//报警复位
IF machine.reset THEN
  MEMSET(ADR(machine.presetAlarms),0,SIZEOF(machine.presetAlarms));
  MEMSET(ADR(machine.userAlarms),0,SIZEOF(machine.userAlarms));
  machine.publicAlarm := FALSE;
  machine.report.alarming := FALSE;
  machine.report.stationAlarming := FALSE;
END_IF;

// 报警顶栏显示
IF NOT alarmingCache AND  machine.alarming THEN
  machine.alarmTopBarDisplay := TRUE;
ELSIF NOT machine.alarming THEN
  machine.alarmTopBarDisplay := FALSE;
END_IF;
alarmingCache :=  machine.alarming;

//复位按钮灯
machine.alarmCanReset := machine.report.alarmCanReset;

machine.resetButtonLight := machine.lampTesthmi        //指示灯测试
OR (NOT machine.alarmCanReset AND machine.alarming) //报警中常亮
OR (machine.alarmCanReset AND clock.c1s);           //报警可复位闪烁
machine.alarmCanReset := FALSE;
machine.report.alarmCanReset := FALSE;
END_ACTION

ACTION AutoTip:
//--------------------------AutoTip---------------------------//
  
//机器未初始化
machine.presetAutoTips[0] := NOT machine.initDone;
//机器运行条件不足
machine.presetAutoTips[1] := NOT machine.runPermit;

//整机自动提示
machine.autoTip :=
FUN_AryBitCount_RD(machine.presetAutoTips) >0
OR FUN_AryBitCount_RD(machine.userAutoTips) >0
OR machine.report.autoTip
OR machine.report.stationAutoTip;
machine.report.autoTip := FALSE;
machine.report.stationAutoTip := FALSE; 

//自动提示弹窗
IF machine.autoTip AND machine.start THEN
  machine.autoTipTrigger := TRUE;
  machine.popup := POPUP_AUTO_TIP;
END_IF;
IF machine.popup = 0 THEN
  machine.autoTipTrigger := FALSE;
END_IF;
END_ACTION

ACTION CycleTime:
//--------------------------CycleTime---------------------------//
//机器周期计时,
IF machine.cycleTimeEnd THEN
  machine.cycleTime :=TIME_TO_DINT( cycleTimeTimer.ET);
END_IF;
cycleTimeTimer(IN := machine.cycleTimeStart AND NOT (machine.cycleTimeEnd OR machine.initing),
               PT := T#10M
);
machine.cycleTimeEnd := FALSE;
END_ACTION

ACTION Empty:
//--------------------------Empty---------------------------//
  
//清料条件
emptyPermit := machine.eStop
AND machine.initDone
AND NOT machine.initing;

// 清料完成，延时复位完成信号
IF machine.emptyDone
  AND NOT machine.emptying   //确保清料中断开
  AND NOT machine.running    //确保自动中断开
THEN
  machine.emptyDone := FALSE;
END_IF;

// 清料hmi，弹出清料确认对话框
IF emptyPermit
  AND machine.emptyhmi
THEN
  machine.popup := POPUP_EMPTY_CONFIRM;
END_IF;
// 清料中
IF NOT machine.initing
  AND NOT machine.emptyDone
THEN
  IF machine.emptyConfirm
    AND emptyPermit
  THEN
    machine.emptying := TRUE;
  END_IF;
  
ELSE
  machine.emptying := FALSE;
END_IF;

// 不在清料中且清料完成，弹出清料完成对话框
// 清料完成信号由功能块外部判断清料完成后置位，功能块内部不进行置位
IF NOT machine.emptying
  AND machine.emptyDone
THEN
  machine.popup := POPUP_EMPTY_DONE;
END_IF;
END_ACTION

ACTION Flow:
//--------------------------Flow---------------------------//
//流程监控
FOR index := 0 TO flowNum DO
  IF machine.flow[index].actStep = 999 THEN
    machine.flow[index].uninterrupted := TRUE;
  END_IF;
  //流程上一步记录
  IF machine.flow[index].actStep <> flowStepCache[index] THEN
    machine.flow[index].prevStep := flowStepCache[index];
  END_IF;
  flowStepCache[index] := machine.flow[index].actStep;
  //流程超时计时
flowTimeoutTimer[index](IN := machine.flow[index].timeoutEnable
            AND NOT machine.flow[index].timeoutException
            AND (machine.running OR machine.initing)
            AND machine.flow[index].actStep > 0
            AND machine.flow[index].actStep = flowStepCache[index],
            PT := machine.flow[index].setTimeout,
		  Q=>);
  machine.flow[index].timeoutException := FALSE;
  //流程超时报警置位
IF flowTimeoutTimer[index].Q THEN
    machine.flow[index].timeoutAlarm := TRUE;
    machine.presetAlarms[index + 8] := TRUE;
  ELSIF machine.reset THEN
    machine.flow[index].timeoutAlarm := FALSE;
  END_IF;
END_FOR;
END_ACTION

ACTION General:
//--------------------------General---------------------------//
FUN_UpdateLeftSidebar_RD(machine:=machine,
			  				hmi:=hmi);

//  触摸屏按钮
machine.start := machine.startButton OR hmi.button.start OR machine.starthmi;
machine.stop := machine.stopButton OR hmi.button.stop OR machine.stophmi;
machine.reset := machine.resetButton OR hmi.button.reset OR machine.resethmi;
machine.pause := machine.pauseButton OR hmi.button.pause OR machine.pausehmi;
machine.init := machine.initButton OR hmi.button.init OR machine.inithmi;
manualSwitch := machine.manualSwitch OR hmi.button.manualSwitch;
autoSwitch := machine.autoSwitch OR hmi.button.autoSwitch;
IF manualSwitch OR autoSwitch THEN
  manualModehmi := FALSE;   //实体手自动旋钮复位hmi
  autoModehmi := FALSE;
END_IF;

IF NOT manualModehmiCache AND machine.manualModehmi THEN
	autoModehmi := FALSE;
	manualModehmi := NOT manualModehmi;
END_IF;
manualModehmiCache := machine.manualModehmi;

IF  NOT autoModehmiCache AND machine.autoModehmi THEN
	autoModehmi := NOT autoModehmi;
	manualModehmi := FALSE;
END_IF;
autoModehmiCache := machine.autoModehmi;

//手动模式
machine.manualMode := NOT machine.jogMode
AND (manualSwitch AND NOT autoSwitch
OR NOT manualSwitch AND NOT autoSwitch
AND manualModehmi AND NOT autoModehmi
);
//自动模式
machine.autoMode := NOT machine.jogMode
AND (NOT manualSwitch AND autoSwitch
OR NOT manualSwitch AND NOT autoSwitch
AND NOT manualModehmi AND autoModehmi
);

IF machine.manualMode THEN
  machine.mode := MANUAL_MODE;
ELSIF machine.autoMode THEN
  machine.mode := AUTO_MODE;
ELSE
  machine.mode := UNDEFINED_MODE;
END_IF;

// 三色灯
machine.greenStatusLight := machine.lampTesthmi OR (machine.running AND NOT machine.alarming);
machine.yellowStatusLight := machine.lampTesthmi OR (NOT machine.running AND NOT machine.alarming);
machine.redStatusLight := machine.lampTesthmi OR machine.alarming;
machine.buzzer := machine.alarming AND NOT buzzerTimer.Q;
buzzerTimer(IN := machine.alarming,
             PT := machine.buzzerTime);
END_ACTION

ACTION Init:
//--------------------------Init---------------------------//
// 初始化条件
initPermit := safePermit
AND machine.manualMode
AND NOT machine.alarming;

//初始化确认弹窗
IF machine.init THEN
  IF machine.alarming THEN
    machine.popup := POPUP_INIT_ALARM;
  ELSIF initPermit AND NOT machine.initing THEN
    machine.popup := POPUP_INIT_FAILED;
  END_IF;
END_IF;

 //整机初始化完成
machine.initDone := initDoneTimer.Q
												AND NOT machine.initConfirm
												AND machine.initFlowDone
												AND NOT machine.report.stationNotInitDone;

// 初始化中
IF initPermit
  AND NOT machine.pause
  AND NOT machine.initDone
AND FUN_AryBitCount_RD(machine.userManualTips) =0
THEN
  IF initConfirmCache AND NOT machine.initConfirm THEN
    machine.initing := TRUE;
  END_IF;
ELSE
  machine.initing := FALSE;
END_IF;
initConfirmCache := machine.initConfirm ;  // 初始化确认下降沿

// 初始化延时
initTimer(IN := machine.initing,
           PT := T#10S,
           Q  => );

// 初始化完成延时
initDoneTimer(IN := NOT machine.initConfirm,
               PT := T#10S,
			 Q=>);

// 初始化超时
initTimeoutTimer(IN := machine.initing,
                  PT := machine.initTimeout);

// 初始化按钮灯，初始化中常亮  
machine.initButtonLight := machine.lampTesthmi OR machine.initing;
  
machine.report.stationNotInitDone := FALSE;

 //整机初始化中下降沿
IF  initingCache AND NOT machine.initing THEN
  IF  machine.alarming THEN			// 初始化中报警对话框
    machine.popup := POPUP_INITING_ALARM;	
	ELSIF machine.initDone THEN		// 初始化完成对话框
    machine.popup := POPUP_INIT_DONE;	  
	ELSE												// 初始化失败对话框
    machine.popup := POPUP_INIT_CONFIRM;
  END_IF;	  
END_IF;
initingCache:=machine.initing;
END_ACTION

ACTION LeftSidebar:
//--------------------------LeftSidebar---------------------------//
  //左侧边栏按钮控制

//---------------------------

hmi.button.startLight := machine.startButtonLight;
hmi.button.stopLight := machine.stopButtonLight;
hmi.button.resetLight :=machine.resetButtonLight;
hmi.button.pauseLight :=   machine.pauseButtonLight;
hmi.button.initLight := machine.initButtonLight;
END_ACTION

ACTION ManualTip:
//--------------------------ManualTip---------------------------//
  
// 复位手动提示
IF machine.reset OR Hmi.machineHmi.tipReset THEN
  machine.tipReset := TRUE;
END_IF;
IF machine.tipReset THEN
  MEMSET(ADR(machine.presetAutoTips),0,SIZEOF(machine.presetAutoTips));
  MEMSET(ADR(machine.userAutoTips),0,SIZEOF(machine.userAutoTips));
  MEMSET(ADR(machine.presetManualTips),0,SIZEOF(machine.presetManualTips));
  MEMSET(ADR(machine.userManualTips),0,SIZEOF(machine.userManualTips));	
  //复位提示窗口
  IF machine.popup = 0 THEN
 Hmi.machineHmi.tipReset:=FALSE;	
    machine.tipReset := FALSE; 
  ELSE
    machine.popup := 0;
  END_IF;
END_IF;

//机器手动提示
IF machine.start OR machine.init THEN
  machine.presetManualTips[0] := NOT machine.eStop;     //急停中,无法操作
  machine.presetManualTips[1] := NOT machine.safety;    //安全条件不满足,无法操作
  machine.presetManualTips[2] := NOT machine.allDoorClosed;  //安全门未锁好,无法操作
  machine.presetManualTips[3] := NOT machine.airOn;     //气压不足,无法操作
  IF machine.init THEN
    machine.presetManualTips[4] := NOT machine.manualMode;//不在手动模式,无法操作
  ELSIF machine.start THEN
    machine.presetManualTips[5] := NOT machine.autoMode;  //不在自动模式,无法操作
  END_IF;
END_IF;

//机器手动提示中
machine.manualTip :=
FUN_AryBitCount_RD(machine.presetManualTips) >0
OR FUN_AryBitCount_RD(machine.userManualTips) >0
OR machine.report.stationManualTip
OR machine.report.manualTip;
machine.report.manualTip := FALSE;
machine.report.stationManualTip := FALSE;

// 手动提示弹窗
IF machine.manualTip THEN
  machine.popup := POPUP_MANUAL_TIP;
END_IF;
END_ACTION

ACTION Paused:
//--------------------------Paused---------------------------//
// 暂停中
IF machine.pause THEN
  machine.paused := TRUE;
END_IF;

// 急停、初始化、启动，复位暂停中
IF NOT machine.eStop
  OR machine.initing
  OR machine.start
THEN
  machine.paused := false;
END_IF;

// 暂停按钮灯，暂停中常亮
machine.pauseButtonLight := machine.lampTesthmi  OR machine.paused;
END_ACTION

ACTION Safety:
//--------------------------Safety---------------------------//
  
//急停就绪    
machine.eStop := NOT machine.report.notEstops;
machine.report.notEstops := FALSE;

//安全门就绪 
// machine.allDoorClosed := NOT machine.report.notSafetyDoors;
machine.report.notSafetyDoors := FALSE;

safePermit := machine.eStop
AND machine.allDoorClosed
AND machine.airOn
AND machine.safety;
END_ACTION

ACTION SetUp:
//--------------------------SetUp---------------------------//

  
IF NOT activated THEN
	  activated:=TRUE;
	//赋初始值
	machine.runPermit			:=TRUE;
	machine.startPermit			:=TRUE;
	machine.mainScreenNo 		:= 10; //自定义主画面显示
	machine.initTimeout			:= T#60s; // 初始化超时时间
	machine.idealCycleTime 		:= t#2s;  //理想周期时间
	machine.stopTimeout			:= T#4s; //停止超时时间,理想周期2倍以上时间
	machine.buzzerTime			:= T#3s; // 蜂鸣器持续时间
	machine.requestCountdown 	:=UINT#10;  // HMI请求控制权倒计时
	machine.sidebar.typeData[1]:=1;
	machine.sidebar.typeData[2]:=2;
	machine.sidebar.typeData[5]:=3;
    //流程数量
	flowNum := SIZEOF(machine.flow) -1;
	FOR index:=0 TO flowNum DO
		//machine.flow[index].timeoutEnable	:=FALSE;
	    machine.flow[index].setTimeout			:=T#30s;
	END_FOR;
	
END_IF;
machine.sidebar.typeData[1]:=1;
machine.sidebar.typeData[2]:=2;
machine.sidebar.typeData[5]:=3;
END_ACTION

ACTION Start:
//--------------------------Start---------------------------//
// 运行条件
machine.ready := safePermit
AND machine.runPermit
AND machine.initDone
AND (machine.autoMode OR machine.jogMode)
AND NOT machine.alarming
AND NOT machine.autoTip;
// 运行中
IF machine.ready
  AND NOT machine.pause
  AND NOT machine.paused
  AND NOT machine.stopDone
  AND NOT machine.emptyDone
THEN
  IF machine.autoMode THEN
    IF machine.start
      AND NOT machine.reset
      AND NOT machine.stop
    THEN     //自动模式下按下启动按钮自动中保持
      machine.running := TRUE;
    END_IF;
  ELSIF machine.jogMode
    AND NOT machine.reset
    AND NOT machine.stop
    AND machine.start
  THEN
    machine.running := TRUE;  //寸动模式下按下启动按钮自动中，抬起按钮复位自动中
  ELSE
    machine.running := FALSE;
  END_IF;
ELSE
  machine.running := FALSE;
END_IF;

// 启动按钮灯，运行中常亮，准备就绪时闪烁

machine.startButtonLight := machine.lampTesthmi
OR machine.running
OR (machine.ready AND clock.c1s);
END_ACTION

ACTION Stop:
//--------------------------Stop---------------------------//
// 自动中按停止，置位停止中
IF (machine.stop OR machine.alarming)
  AND NOT machine.stopDone
  AND NOT machine.paused
THEN
  machine.stopping := TRUE;
END_IF;

// 急停，初始化，启动，暂停，停止完成且不在自动中，复位停止中
IF NOT machine.eStop
  OR machine.initing
  OR machine.start
  OR machine.pause
  OR machine.stopDone
  AND NOT machine.running
THEN
  machine.stopping := FALSE;
END_IF;

//停止完成
stopTimer(IN := machine.stopping,
           PT := machine.stopTimeout);
IF machine.stopping AND (machine.stopDoneAllow OR stopTimer.Q) THEN
  machine.stopDone := TRUE;
ELSIF NOT machine.eStop
  OR machine.initing
  OR machine.start
  OR machine.pause
THEN
  machine.stopDone := FALSE;
END_IF;

// 停止按钮灯，停止完成常亮，停止中闪烁
  machine.stopButtonLight := machine.lampTesthmi
OR machine.stopDone
OR (machine.stopping AND clock.c1s);
END_ACTION

ACTION Tip:
//--------------------------Tip ---------------------------//
  
IF machine.alarming THEN
  machine.status := ALARMING;
ELSIF machine.initing THEN
  machine.status := INITING;
ELSIF machine.running THEN
  machine.status := RUNNING;
ELSIF machine.ready THEN
  machine.status := READY;
ELSE
  machine.status := 0;
END_IF;

machine.presetTips[1] := machine.alarming;
machine.presetTips[2] := machine.paused;
machine.presetTips[3] := machine.stopping;
machine.presetTips[4] := machine.initing;
machine.presetTips[5] := machine.running;
machine.presetTips[6] := machine.ready AND NOT machine.running;
machine.presetTips[7] := NOT machine.ready;
machine.presetTips[10] := machine.emptying;
machine.presetTips[11] := machine.emptyDone;
machine.presetTips[21] := machine.dryRun;
END_ACTION

END_FUNCTION_BLOCK

// ---- Standard/FUN/FUN_UpdateLeftSidebar_RD.TcPOU
FUNCTION FUN_UpdateLeftSidebar_RD : bool
VAR_IN_OUT
machine       : UDT_Machine_RD;
hmi           : UDT_hmi_RD;
END_VAR
VAR CONSTANT
LEFT_SIDEBAR_MANUAL_MODE : INT :=1;
LEFT_SIDEBAR_AUTO_MODE   : INT :=2;
LEFT_SIDEBAR_JOG_MODE    : INT :=3;
LEFT_SIDEBAR_SETUP_MODE  : INT :=4;
LEFT_SIDEBAR_INIT        : INT :=5;
LEFT_SIDEBAR_START       : INT :=6;
LEFT_SIDEBAR_STOP        : INT :=7;
LEFT_SIDEBAR_RESET       : INT :=8;
LEFT_SIDEBAR_EMPTY       : INT :=9;
LEFT_SIDEBAR_PAUSE       : INT :=10;
LEFT_SIDEBAR_MANUAL      : INT :=11;
LEFT_SIDEBAR_PARAMETER   : INT :=12;
LEFT_SIDEBAR_STATION     : INT :=13;

END_VAR

// 获取左侧边栏按钮是否按下
machine.manualModeHmi := machine.sidebar.click[LEFT_SIDEBAR_MANUAL_MODE];
machine.autoModeHmi := machine.sidebar.click[LEFT_SIDEBAR_AUTO_MODE];
machine.jogModeHmi := machine.sidebar.click[LEFT_SIDEBAR_JOG_MODE];
machine.setupModeHmi := machine.sidebar.click[LEFT_SIDEBAR_SETUP_MODE];
machine.initHmi := machine.sidebar.click[LEFT_SIDEBAR_INIT];
machine.startHmi := machine.sidebar.click[LEFT_SIDEBAR_START];
machine.stopHmi := machine.sidebar.click[LEFT_SIDEBAR_STOP];
machine.resetHmi := machine.sidebar.click[LEFT_SIDEBAR_RESET];
machine.emptyHmi := machine.sidebar.click[LEFT_SIDEBAR_EMPTY];
machine.pauseHmi := machine.sidebar.click[LEFT_SIDEBAR_PAUSE];
IF machine.sidebar.click[LEFT_SIDEBAR_MANUAL] THEN
	hmi.toManualPageClick:=TRUE;
END_IF;
IF machine.sidebar.click[LEFT_SIDEBAR_PARAMETER] THEN
	hmi.toParameterPageClick:=TRUE;
END_IF;
IF machine.sidebar.click[LEFT_SIDEBAR_STATION] THEN
	hmi.toStationPageClick:=TRUE;
END_IF;

// 设置左侧边栏按钮状态显示
machine.sidebar.status[LEFT_SIDEBAR_MANUAL_MODE] := machine.manualMode;
machine.sidebar.status[LEFT_SIDEBAR_AUTO_MODE] := machine.autoMode;
machine.sidebar.status[LEFT_SIDEBAR_JOG_MODE] := machine.jogMode;
machine.sidebar.status[LEFT_SIDEBAR_SETUP_MODE] := machine.setupMode;
machine.sidebar.status[LEFT_SIDEBAR_INIT] := machine.initButtonLight;
machine.sidebar.status[LEFT_SIDEBAR_START] := machine.startButtonLight;
machine.sidebar.status[LEFT_SIDEBAR_STOP] := machine.stopButtonLight;
machine.sidebar.status[LEFT_SIDEBAR_RESET] := machine.resetButtonLight;
machine.sidebar.status[LEFT_SIDEBAR_EMPTY] := machine.emptying;
machine.sidebar.status[LEFT_SIDEBAR_PAUSE] := machine.pauseButtonLight;
machine.sidebar.status[LEFT_SIDEBAR_MANUAL] := hmi.inManualPage;
machine.sidebar.status[LEFT_SIDEBAR_PARAMETER] := hmi.inParameterPage;
machine.sidebar.status[LEFT_SIDEBAR_STATION] := hmi.inStationPage;

END_FUNCTION

// ---- Standard/Unit/03 Estop/FB_Estop_RD.TcPOU
FUNCTION_BLOCK FB_Estop_RD
VAR_IN_OUT
vari         : UDT_Estop_RD;
machine      : UDT_Machine_RD;

END_VAR
VAR
resetCache      : BOOL;
END_VAR

//急停复位
IF machine.reset AND NOT resetCache AND vari.input THEN
	vari.notEstop:=FALSE;
END_IF;

//急停
IF NOT vari.disable AND NOT vari.input THEN
	Vari.notEstop:=TRUE;
	machine.report.notEstops:=TRUE;
END_IF;

resetCache:=machine.reset;

END_FUNCTION_BLOCK

// ---- Standard/Unit/04 SafetyDoor/FB_SafetyDoor_RD.TcPOU
FUNCTION_BLOCK FB_SafetyDoor_RD
VAR_IN_OUT
machine : UDT_Machine_RD; //
vari : UDT_SafetyDoor_RD; //
clock : UDT_Clock_RD; //
END_VAR

VAR
prohibit : BOOL; // 禁止解锁
unlockButtonCache : Bool; // 解锁按钮缓存
permitTimer : TON; // 解锁许可延时
autoLockTimer : TON; // 自锁延时

END_VAR

VAR CONSTANT
NOT_LOCKED      : UINT:=1;
DISABLED        : UINT:=2;
END_VAR

  //================================================================================== 
  // Harmontromics / (C) Copyright (2021) 
  //----------------------------------------------------------------------------------
  // Title:               Safety Door
  // Comment/Function:    实现安全门的控制，自/手动上锁、按钮解锁
  // Library/Family:      (that the source is dedicated to)
  // Author:              David.Wong
  // Target System: 
  // Engineering:         Sysmac Studio
  // Restrictions:        (OB types, etc.)
  // Requirements:        (hardware, technological package, etc.) 
  //----------------------------------------------------------------------------------
  // Change log table:
  // Version     | Date       | Expert in charge | Changes applied
  //-------------|------------|------------------|------------------------------------
  // 001.000.000 | 2021-12-11 | David.Wong       | First released version
  //             |            |                  | 
  //             |            |                  |              
  //             |            |                  | 
  //================================================================================== 
SetUp();
SafetyDoor();
Tip();

ACTION SafetyDoor:
//------------------------------SafetyDoor-------------------------------------//
  
//  禁止解锁
prohibit := machine.eStop
AND vari.inputLocked
AND (NOT machine.manualMode
OR machine.initing
OR machine.running
OR vari.prohibitUnlock);

//  解锁许可延时
permitTimer(
	IN:=NOT Prohibit,
	PT:=T#500MS,
	Q=> , ET=> 
);
  
//  插销没到位且没锁好信号时自动弹开
IF vari.inputUnlockButton
	AND
	permitTimer.Q	  
	//AND NOT vari.inputLocked   
	//AND NOT vari.inputArrived
THEN
  vari.outputLockCoil := TRUE;
END_IF;

//  解锁按钮操作，自动上锁时解锁，非自动上锁时解锁和上锁
IF NOT unlockButtonCache AND vari.inputUnlockButton THEN
  vari.outputLockCoil := NOT vari.outputLockCoil AND NOT vari.autoLock;
END_IF;
unlockButtonCache := vari.inputUnlockButton;

//  自锁延时
autoLockTimer(IN := vari.autoLock AND NOT vari.inputUnlockButton,
			  PT := vari.autoLockTime
);  
  
//  自动上锁及禁止解锁
IF vari.inputArrived
  AND
  (autoLockTimer.Q
  OR NOT permitTimer.Q)
THEN
  vari.outputLockCoil := FALSE;
END_IF;

//  解锁按钮灯输出
IF vari.inputLocked THEN
  vari.outputUnlockButtonLight := vari.lightWhenLocked;
ELSE
  vari.outputUnlockButtonLight := clock.c1s;
END_IF;
END_ACTION

ACTION SetUp:
//------------------------------SetUp-------------------------------------//
  IF machine.startUp THEN
    IF vari.name[machine.actLanguage] <> '' THEN
      vari.name[0] := vari.name[machine.actLanguage];
    END_IF;
	vari.autoLockTime:=T#3s;
  END_IF;
END_ACTION

ACTION Tip:
//------------------------------Tip---------------------------------------------//
  
// 安全门未锁好提示
IF (NOT vari.inputArrived
  OR NOT vari.inputLocked
  OR NOT vari.outputLockCoil)
  AND NOT vari.disabled
THEN
  vari.notLocked := TRUE; // 安全门未锁好报警
ELSIF machine.reset THEN
  vari.notLocked := FALSE;
END_IF;

//反馈安全没锁好
IF vari.notLocked THEN
  machine.report.notSafetyDoors := TRUE;
END_IF;
END_ACTION

END_FUNCTION_BLOCK

// ---- Standard/Unit/07 Sensor/FB_Sensor_RD.TcPOU
FUNCTION_BLOCK FB_Sensor_RD
VAR_IN_OUT
machine : UDT_Machine_RD; //
station : UDT_Station_RD; //
vari : UDT_SensorVar_RD; //
data : UDT_SensorData_RD; //
END_VAR
VAR_OUTPUT
END_VAR
VAR
inputCache : BOOL; //
checkCache : Bool; //
resetCache : Bool; //
onTimer : TON; //
offTimer : TON; //
flickerTimer : TON; //
firstCall    : BOOL :=TRUE;

END_VAR

SetUp();
Delay();
Alarm();

ACTION Alarm:
//-------------------------------Alarm--------------------------//
  
//复位报警并计数清零
IF NOT resetCache AND machine.reset THEN
  IF vari.unchangeError THEN
    vari.count := 0;
    vari.unchangeError := FALSE;
  END_IF;
  vari.flickerError := FALSE;
END_IF;
resetCache := machine.reset;
  
vari.alarming := vari.unchangeError
OR vari.flickerError;

//反馈上一级报警中
IF vari.alarming THEN
  station.report.alarming := TRUE;
  machine.alarmCount := machine.alarmCount +1;
END_IF;
END_ACTION

ACTION Delay:
//-----------------------------------Delay--------------------------//
//屏蔽传感器时,ON OFF都输出
IF NOT data.disabled THEN
  onTimer(IN := vari.input,
           PT :=UDINT_TO_TIME(data.onTime),
           Q => vari.isOn);
  offTimer(IN := NOT vari.input,
            PT := UDINT_TO_TIME(data.offTime),
            Q => vari.isOff);
  IF inputCache <> vari.input OR data.setCount = 0 THEN//输入有变化或设置值0清空计数
    vari.count := 0;
  ELSIF NOT checkCache AND vari.check THEN    //check上升沿计数+1
    vari.count :=vari.count + 1;
  ELSIF checkCache AND NOT vari.check       //check下降沿且计数计数值大于等于设定值时报警
    AND vari.count >= data.setCount
  THEN
    vari.unchangeError := TRUE;
  END_IF;
  
  //超过On、Off延时之和2倍时间都没到位报警传感器闪烁异常
  data.flickerTime := MAX(data.flickerTime,(data.onTime + data.offTime) * 2);
  flickerTimer(IN := NOT vari.isOn AND NOT vari.isOff,
               PT := UDINT_TO_TIME(data.flickerTime)
			   );
  
  inputCache := vari.input;
  checkCache := vari.check;
ELSE
  vari.isOn := TRUE;
  vari.isOff := TRUE;
  vari.count := 0;
END_IF;
END_ACTION

ACTION SetUp:
//开机或切换语言后执行一个扫描周期
//------------------------------------ SetUp--------------------------//
  IF firstCall THEN
    // 显示在HMI上面
    vari.display := TRUE;
	firstCall :=FALSE;
  END_IF;
END_ACTION

END_FUNCTION_BLOCK

// ---- Standard/Unit/12 Delay/FB_Delay_RD.TcPOU
FUNCTION_BLOCK FB_Delay_RD
VAR_IN_OUT
machine : UDT_Machine_RD; //
station : UDT_Station_RD; //
vari : UDT_DelayVar_RD; //
data : UDT_DelayData_RD; //
END_VAR
VAR_OUTPUT
END_VAR

VAR
timer1    : TON;
END_VAR

timer1(IN := vari.input AND vari.actTime <= data.setTime,
	         PT := data.setTime,
	         ET => vari.actTime,
	         Q => vari.isOn);
IF vari.isOn OR vari.actTime > data.setTime THEN
  vari.input := FALSE;
END_IF;

END_FUNCTION_BLOCK

// ---- Standard/Unit/08 Motor/FB_Motor_RD.TcPOU
FUNCTION_BLOCK FB_Motor_RD
VAR_IN_OUT
machine   : UDT_Machine_RD;
station   : UDT_Station_RD;
vari      : UDT_MotorVar_RD;
data      : UDT_MotorData_RD;
END_VAR
VAR
forwardAllow : BOOL; // 正转允许
reversalAllow : Bool; // 反转允许
safetyPermit : Bool; // 安全条件
resetCache : Bool; // 复位缓存
forwardHmiCache : Bool; // 正转Hmi缓存
reverseHmiCache : Bool; // 反转Hmi缓存
veeredTimer : TON; // 正反转切换延时器
veeredTimer2 : TON; // 正反转切换延时器
startTimer : TON; // 启动延时器
forwardStopTimer : TON; // 正转停止延时器
reversalStopTimer : TON; // 反转停止延时器
runMonitorTimer : TON; // 运行监控延时器
forwardMode : Bool; // 正转模式
reversalMode : Bool; // 反转模式
pushAlarmNo : UInt; //
pushManualTipNo : UInt; //
pushAutoTipNo : UInt; //
activated : BOOL; //

END_VAR

VAR CONSTANT
OFF_STATE : UINT:=0; // OFF状态
ON_STATE : UINT:=1; // ON状态
INOPERABLE_STATE : UINT:=2; // 不可操作状态
ENABLE_RUN_MONITOR : UINT:=1; // 启用运行监控
INVERTER_ALARM : UINT:=1; // 变频器报警
NOT_FEEDBACK_ALARM : UINT:=2; // 无运行反馈报警
AUTO_TIP : UINT:=3; // 手动操作中自动提示
NO_FORWARD_PERMIT : UINT:=4; // 正转动作条件不满足
NO_REVERSAL_PERMIT : UINT:=5; // 反转动作条件不满足
END_VAR

//------------------------Description header 
  //================================================================================== 
  // Harmontromics / (C) Copyright (2021) 
  //----------------------------------------------------------------------------------
  // Title:               Motor Control
  // Comment/Function:    普通交流电机的正向/反向控制，运行监控以及错误报警
  // Library/Family:      瀚川标准库
  // Author:              David.Wong
  // Target System:       无
  // Engineering:         TIA Portal (V15.1)
  // Restrictions:        无
  // Requirements:        无
  //----------------------------------------------------------------------------------
  // Change log table:
  // Version     | Date       | Expert in charge | Changes applied
  //-------------|------------|------------------|------------------------------------
  // 001.000.000 | 2021-12-11 | David.Wong       | 首次发布的版本
  // 001.000.001 | 2021-12-24 | David.Wong       | 增加启动-停止延迟
  // 001.001.001 | 2022-4-29  | David.Wong       | 增加运行监控和错误报警          
  // 002.000.001 | 2023-6-9   | David.Wong       | 增加启动完成延时
  //             |            |                  |
  //================================================================================== 
SetUp();
Alarm();
General();
Manual();
Auto();
ManualTip();
AutoTip();
Status();
Output();
Cache();

ACTION Alarm:
//------------------------Alarm------------------------//

//报警复位
IF NOT resetCache AND machine.reset THEN
  vari.inverterAlarm := FALSE;
  vari.runningAlarm := FALSE;
END_IF;

//变频器复位
vari.outputErrorReset := vari.inputError AND machine.reset;

//变频器错误
IF vari.inputError THEN
  vari.inverterAlarm := TRUE;
END_IF;

//运行反馈错误
IF vari.monitorMode = ENABLE_RUN_MONITOR THEN
  runMonitorTimer(IN := (vari.outputReversal OR vari.outputForward) XOR vari.inputRunning,		  				
			PT := T#30S,
			Q=>	);
  IF runMonitorTimer.Q THEN
    vari.runningAlarm := TRUE;
  END_IF;
ELSE
  vari.inputRunning := vari.outputReversal OR vari.outputForward;
END_IF;


//报警中
vari.alarming := vari.inverterAlarm OR vari.runningAlarm;
//反馈上级报警中
IF vari.alarming THEN
  station.report.alarming := TRUE;
  machine.alarmCount := machine.alarmCount +1;
END_IF;
END_ACTION

ACTION Auto:
//------------------------Auto------------------------//
  
  // 启动和停止延时
  	startTimer(IN := vari.outputForward OR vari.outputReversal,		
			PT := DINT_TO_TIME(data.startTime),
			Q=>	);
  IF startTimer.Q AND NOT vari.alarming THEN
    vari.inForward := vari.outputForward;
    vari.inReversal := vari.outputReversal;
  ELSE
    vari.inForward := FALSE;
    vari.inReversal := FALSE;
  END_IF;
	forwardStopTimer(IN := vari.forwardManual = vari.forwardAuto,			
			PT := DINT_TO_TIME(data.stopTime),
			Q=>);
	reversalStopTimer(IN := vari.reversalManual = vari.reversalAuto,
		PT := DINT_TO_TIME(data.stopTime) ,
		Q=>);
END_ACTION

ACTION AutoTip:
//------------------------AutoTip------------------------//
  
//自动提示
vari.autoTip := vari.forwardManual OR vari.reversalManual;
IF vari.autoTip
  AND (station.autoTipTrigger OR machine.autoTipTrigger)
THEN
  pushAutoTipNo := AUTO_TIP;
ELSE
  pushAutoTipNo := 0;
END_IF;

//反馈工站自动提示
IF vari.autoTip THEN
  station.report.autoTip := TRUE;
END_IF;
END_ACTION

ACTION Cache:
//------------------------Cache------------------------//
  
resetCache := machine.reset;
forwardHmiCache := vari.forwardHmi;
reverseHmiCache := vari.reversalHmi;
vari.init := FALSE;
END_ACTION

ACTION General:
//------------------------General ------------------------//
  
//安全条件
safetyPermit := machine.eStop
AND machine.safety
AND machine.allDoorClosed;

//正反转模式
forwardMode := vari.turnMode = 1 OR vari.turnMode = 3;
reversalMode := vari.turnMode = 2 OR vari.turnMode = 3;

//正转允许操作
IF safetyPermit
  AND NOT vari.alarming
THEN
  forwardAllow := forwardMode AND vari.forwardPermit;
  reversalAllow := reversalMode AND vari.reversalPermit;
ELSE
  forwardAllow := FALSE;
  reversalAllow := FALSE;
END_IF;
END_ACTION

ACTION Manual:
//------------------------Manual------------------------//
  
IF machine.manualMode
  AND NOT vari.init
THEN
  vari.forwardForbidIcon := forwardMode AND NOT forwardAllow;
  vari.reversalForbidIcon := reversalMode AND NOT reversalAllow;
  //正转手动操作
  IF forwardAllow THEN
    IF forwardHmiCache AND NOT vari.forwardHmi THEN
      vari.forwardManual := NOT vari.forwardManual;
      vari.reversalManual := FALSE;
    END_IF;
  ELSE
    vari.forwardManual := FALSE;
  END_IF;
  
  //反转手动操作
  IF reversalAllow THEN
    IF reverseHmiCache AND NOT vari.reversalHmi THEN
      vari.reversalManual := NOT vari.reversalManual;
      vari.forwardManual := FALSE;
    END_IF;
  ELSE
    vari.reversalManual := FALSE;
  END_IF;
  
ELSE
  vari.forwardManual := FALSE;
  vari.reversalManual := FALSE;
  vari.forwardForbidIcon := forwardMode;
  vari.reversalForbidIcon := reversalMode;
END_IF;
END_ACTION

ACTION ManualTip:
//------------------------ManualTip------------------------//
  
IF machine.tipReset THEN
  vari.forwardManualTip := FALSE;
  vari.reversalManualTip := FALSE;
ELSIF vari.forwardHmi AND forwardMode
  OR vari.reversalHmi AND reversalMode
THEN
  machine.presetManualTips[0] := NOT machine.eStop;     //急停中,无法操作
  machine.presetManualTips[1] := NOT machine.safety;    //安全条件不满足,无法操作
  machine.presetManualTips[2] := NOT machine.allDoorClosed;  //安全门未锁好,无法操作
  machine.presetManualTips[4] := NOT machine.manualMode;//不在手动模式,无法操作
  
  IF safetyPermit AND machine.manualMode THEN
    IF NOT vari.forwardPermit AND vari.forwardHmi THEN
      vari.forwardManualTip := TRUE;//正转条件不满足，用于置位外部提示信息用
    ELSIF NOT vari.reversalPermit AND vari.reversalHmi THEN
      vari.reversalManualTip := TRUE;//反转条件不满足，用于置位外部提示信息用
    END_IF;
  END_IF;
  
END_IF;

//反馈工站手动提示
IF vari.forwardManualTip
  OR vari.reversalManualTip
THEN
  station.report.manualTip := TRUE;
END_IF;
END_ACTION

ACTION Output:
//------------------------Output  ------------------------//
	veeredTimer(IN := NOT vari.outputReversal,
		  PT := T#5S,
		  Q=>);
  	veeredTimer2(IN := NOT vari.outputReversal,
		  PT := T#5S,
		  Q=>);
vari.outputForward := veeredTimer.Q
AND (
(vari.forwardManual XOR vari.forwardAuto)
OR (vari.outputForward AND NOT forwardStopTimer.Q)
);

vari.outputReversal := veeredTimer2.Q
AND (
(vari.reversalManual OR vari.reversalAuto)
OR (vari.outputReversal AND NOT reversalStopTimer.Q)
);
END_ACTION

ACTION SetUp:
//------------------------SetUp------------------------//
  
IF NOT activated THEN
  activated:=TRUE;
  // 赋初始值
vari.forwardPermit		:=TRUE;
vari.reversalPermit		:=TRUE;
vari.turnMode				:=1;

END_IF;
END_ACTION

ACTION Status:
//------------------------Status------------------------//
  
//正转钮指示状态
IF forwardMode THEN
  IF vari.forwardManual THEN
    vari.forwardHmiState := ON_STATE;
  ELSE
    vari.forwardHmiState := OFF_STATE;
  END_IF;
ELSE
  vari.forwardHmiState := INOPERABLE_STATE;
END_IF;

//反转钮指示状态
IF reversalMode THEN
  IF vari.reversalManual THEN
    vari.reversalHmiState := ON_STATE;
  ELSE
    vari.reversalHmiState := OFF_STATE;
  END_IF;
ELSE
  vari.reversalHmiState := INOPERABLE_STATE;
END_IF;
END_ACTION

END_FUNCTION_BLOCK

// ---- Standard/Public/08 WearPart/FB_WearPart.TcPOU
FUNCTION_BLOCK FB_WearPart
VAR_INPUT
localClock : DATE_AND_TIME; //
END_VAR
VAR_IN_OUT
machine : UDT_Machine_RD; //
stations : UDT_Station_RD; //
vari : UDT_WearPartVar_RD; //
data : UDT_WearPartData_RD; //
END_VAR
VAR
nIndex : UINT;
tipTimes : DINT;//提示次数             
END_VAR

Execute();
Alarm();
Clear();

ACTION Alarm:
tipTimes:=LREAL_TO_DINT(DINT_TO_LREAL(data.maxUsage)*REAL_TO_LREAL(data.tipRate)/100);


vari.alarming:=data.actUsage>=data.maxUsage;
vari.tip:=data.actUsage>=tipTimes AND NOT vari.alarming;
END_ACTION

ACTION Clear:
vari.clearHmi :=
vari.clearAuto := FALSE;
IF data.actUsage>0 THEN
  vari.clearAllow:=vari.clearPermit;
  IF vari.clearAllow AND machine.manualMode THEN
      vari.clearForbidIcon := NOT vari.clearAllow;//清零禁止图标
      IF vari.clearAllow AND (vari.clearHmi OR  vari.clearAuto) THEN
        FOR nIndex:=9 TO 1 BY -1 DO
  		  data.recordsTime[nIndex]:=data.recordsTime[nIndex-1];
  		  data.recordsUsage[nIndex]:=data.recordsUsage[nIndex-1];
  	    END_FOR
  	    data.recordsTime[0]:=DT_TO_SYSTEMTIME(localClock);
  	    data.recordsUsage[0]:=data.actUsage;
  	    data.actUsage:=0;
      END_IF;
  ELSE
    vari.clearForbidIcon := TRUE;
  END_IF;
END_IF
END_ACTION

ACTION Execute:
vari.countExecute:=FALSE;
IF vari.countExecute THEN
	data.actUsage:=data.actUsage+vari.increments;
END_IF
END_ACTION

END_FUNCTION_BLOCK

// ---- Standard/Public/11 Oee/FB_Oee_RD.TcPOU
FUNCTION_BLOCK FB_Oee_RD
VAR_INPUT
localClock : DATE_AND_TIME; //
END_VAR
VAR_OUTPUT
END_VAR

VAR_IN_OUT
vari : UDT_OeeVar_RD; //
data : UDT_OeeData_RD; //
lastData : UDT_OeeData_RD; //
END_VAR

VAR
startCache : BOOL; //
endCache : Bool; //
clearCache : Bool; //
failureCache : Bool; //
goodValueCache : DInt; //
badValueCache : DInt; //
secondCache : DATE_AND_TIME; //
nTimer		: UDINT;//计时器，单位100ns，除于10000后单位ms
IdealProducts : DInt; //
emptyData : UDT_OeeData_RD; //
CurTaskInfo	: PlcTaskSystemInfo;//当前任务信息
failureR_Trig   : R_TRIG;
END_VAR

Cache();
Count();
Refresh();
StartEnd();
Timer();

ACTION Cache:
//----------------------Cache--------------------//
failureR_Trig(CLK:=vari.keep AND NOT vari.scheduledDown AND vari.alarming);

goodValueCache := vari.goodValue;
badValueCache := vari.badValue;
secondCache := localClock;
failureCache := vari.keep AND NOT vari.scheduledDown AND vari.alarming;
startCache := vari.start;
endCache := vari.end;
clearCache := vari.clear;
vari.start := FALSE;
vari.end := FALSE;
vari.clear := FALSE;
END_ACTION

ACTION Count:
 //----------------------Count--------------------//
 //OEE统计开始/结束
IF vari.keep OR vari.end THEN
	
    //良品数量增加时，OEE统计会对增加部分累计加
    IF vari.goodValue > goodValueCache THEN
      data.goodValue 	:= data.goodValue + (vari.goodValue - goodValueCache);
      data.totalValue	 	:= data.totalValue +(vari.goodValue - goodValueCache);
    END_IF;
    //不良品数量增加时，OEE统计会对增加部分累计加
    IF vari.badValue > badValueCache THEN
      data.badValue 	:= data.badValue + (vari.badValue - badValueCache);
      data.totalValue 	:= data.totalValue + (vari.badValue - badValueCache);
    END_IF;
    
    //产生故障上升沿增加1次
    IF failureR_Trig.Q THEN
      data.failureCount := data.failureCount +1;
    END_IF;
END_IF
END_ACTION

ACTION Refresh:
//----------------------Refresh--------------------//
//OEE统计开始/结束
IF vari.keep OR vari.end THEN
	//每秒钟运行一次
    IF TRUE THEN
      FUN_TimeToDate_RD(InOut:=data.totalTime);
	  FUN_TimeToDate_RD(InOut:=data.productiveTime);
	  FUN_TimeToDate_RD(InOut:=data.downTime);
	  FUN_TimeToDate_RD(InOut:=data.runtime);
	  FUN_TimeToDate_RD(InOut:=data.standbyTime);
	  FUN_TimeToDate_RD(InOut:=data.failureTime);
	
      
      //时间利用率
      IF data.productiveTime.timeValue > 0 THEN
        data.availability :=  LREAL_TO_REAL(UDINT_TO_LREAL(data.runtime.timeValue)/ UDINT_TO_LREAL(data.productiveTime.timeValue)) * 100;
      ELSE
        data.availability := 0.0;
      END_IF
      
      //性能
      IF vari.idealCycleTime > T#0MS THEN
        IdealProducts := UDINT_TO_DINT(data.runtime.timeValue) / TIME_TO_DINT(vari.idealCycleTime);
        IF IdealProducts > 0 THEN
          data.performance := DINT_TO_REAL(data.totalValue)  / DINT_TO_REAL(IdealProducts)* 100.0;
        ELSE
          data.performance := 0.0;
        END_IF
      ELSE
        IdealProducts := 0;
        data.performance := 0.0;
      END_IF
      
      //质量
      IF data.totalValue > 0 THEN
        data.quality := 100.0 * DINT_TO_REAL(data.goodValue) / DINT_TO_REAL(data.totalValue);
      ELSE
        data.quality := 0.0;
      END_IF
      
      //OEE
      data.oee := (data.availability * data.performance * data.quality) / 10000.0;
      
    END_IF
  
END_IF
END_ACTION

ACTION StartEnd:
//----------------------Start End--------------------//
  
//OEE统计开始/结束
IF NOT startCache AND vari.start THEN
  IF NOT vari.keep THEN
    data := emptyData;  //清空数据
    data.startTime := localClock; //开始时刻
    data.startTimeDisplay := TRUE;
    vari.keep := TRUE;
  END_IF
  vari.scheduledDown := FALSE; //复位计划停机
ELSIF NOT endCache AND vari.end THEN
  IF vari.keep THEN
    data.endTime := localClock; //结束时刻
    data.endTimeDisplay := TRUE;
    lastData := data; //数据存入上一次数据中
    vari.keep := FALSE;
  END_IF
END_IF
  


//清空数据
IF NOT vari.keep
  AND NOT clearCache
  AND  vari.clear
THEN
  data := emptyData;
END_IF
END_ACTION

ACTION Timer:
//----------------------Timer--------------------//
//OEE统计开始/结束
IF vari.keep OR vari.end THEN
	nTimer:=nTimer
		+ MAX(CurTaskInfo.CycleTime, CurTaskInfo.LastExecTime);
END_IF
IF nTimer >= 10000000 THEN
	IF vari.keep
	THEN
		data.totalTime.timeValue:= data.totalTime.timeValue+1;
	END_IF
	
	IF vari.keep AND vari.scheduledDown
	THEN
		data.downTime.timeValue:= data.downTime.timeValue+1;
	END_IF
	
	IF vari.keep AND NOT vari.scheduledDown
	THEN
		data.productiveTime.timeValue:= data.productiveTime.timeValue+1;
	END_IF
	
	IF vari.keep AND NOT vari.scheduledDown AND vari.running
	THEN
		data.runtime.timeValue:= data.runtime.timeValue+1;
	END_IF
	
	IF vari.keep AND NOT vari.scheduledDown AND NOT vari.running AND NOT vari.alarming
	THEN
		data.standbyTime.timeValue:= data.standbyTime.timeValue+1;
	END_IF
	
	IF vari.keep AND NOT vari.scheduledDown AND vari.alarming
	THEN
		data.failureTime.timeValue:= data.failureTime.timeValue+1;
	END_IF
	nTimer:=nTimer - 10000000;
END_IF
END_ACTION

END_FUNCTION_BLOCK

// ---- Standard/FUN/FUN_TimeToDate_RD.TcPOU
FUNCTION FUN_TimeToDate_RD : bool
VAR_IN_OUT
	InOut          : UDT_DayTime_RD;
END_VAR

//	时间转换
InOut.day:=UDINT_TO_USINT(
	InOut.timeValue / 86400
);
InOut.hour:=UDINT_TO_USINT(
	(InOut.timeValue / 3600) MOD 24
);
InOut.minute:=UDINT_TO_USINT(
	(InOut.timeValue / 60) MOD 60
);
InOut.second:=UDINT_TO_USINT(
	InOut.timeValue MOD 60
);

END_FUNCTION

// ---- Standard/Unit/11 KeyenceScan/FB_KeyenceScan_RD.TcPOU
FUNCTION_BLOCK FB_KeyenceScan_RD
VAR_IN_OUT
machine : UDT_Machine_RD; //
station : UDT_Station_RD; //
vari : UDT_KeyenceScanVar_RD; //
data : UDT_KeyenceScanData_RD; //
END_VAR
VAR_OUTPUT
END_VAR
VAR
activated : BOOL; // 块已运行
moduleType : UINT; // 模块类型 0:N-L20, 1:SR-1000X, 2:SR-2000X, 3:SR-LR1
triggerStep : UInt; // 流程字
resetCache : Bool; // 复位缓存
triggerAutoCache : Bool; // 触发Auto缓存
triggerHmiCache : Bool; // 触发Hmi缓存
gradeCache : Int; // ISO_IEC_16022等级缓存
readRequest : Bool; // 读取请求
errorClear : Bool; // 错误清除
readCompleteClear : Bool; // 读取完成清除
error : Bool; //错误
allbusy : Bool; //忙
trgBusy : Bool; //触发忙
readComplete : Bool; //读取完成
resultDataSize : UInt; // 结果数据大小
generalErrorCode : UInt; // 一般错误代码
resultData : Array[0..256] of Byte; // 结果数据
ISO_IEC15415Grade : UInt; // ISO/IEC15415等级
ISO_IEC_TR29158Grade : UINT; // ISO/IEC TR 29158等级
timeoutTimer : TON; //
isTimeoutTimer : BOOL; //
index          : UINT;
END_VAR

VAR CONSTANT
ISO_IEC_15415 	 : UINT :=1 ; // 扫码等级评估标准
ISO_IEC_TR_29158 : UINT :=2 ; // 扫码等级评估标准
ISO_IEC_16022    : UINT :=3 ; // 扫码等级评估标准
RESULT_PASS      : UINT :=1 ; // 扫码结果Pass
RESULT_FAIL      : UINT :=2 ; // 扫码结果Fail
RESULT_TIMEOUT   : UINT :=3 ; // 扫码结果Timeout
ERR_GENERAL      : UINT :=1 ; // 一般错误
ERR_READL 		 : UINT :=2 ; // 读取错误
ERR_TIMEOUT      : UINT :=3 ; // 超时报警
BUSY             : UINT :=4 ; // 处理中
READ_SUCCESS     : UINT :=6 ; // 读取完成
READY            : UINT :=7 ; // 准备就绪
LEVEL_INVALID    : UINT :=99 ; // 扫码等级无效
LEVEL_A 		 : UINT :=4 ; // 扫码等级A
LEVEL_B          : UINT :=3 ; // 扫码等级B
LEVEL_C          : UINT :=2 ; // 扫码等级C
LEVEL_D 		 : UINT :=1 ; // 扫码等级D
LEVEL_F 		 : UINT :=0 ; // 扫码等级F
N_L21 			 : UINT :=0 ; //
SR_1000X 		 : UINT :=1 ; //
SR_2000X 		 : UINT :=2 ; //
SR_LR1 			 : UINT :=3 ; //
END_VAR

SetUp();
InPutUpdate();
Alarm();
General();
ScanFlow();
ManualTip();
OutPutUpdate();
Cache();

ACTION Alarm:
//-----------------------------------------Alarm-----------------------------------------//  
//报警复位
IF NOT resetCache AND machine.reset THEN
  vari.generalError := FALSE;
  vari.readError := FALSE;
  vari.readTimeoutAlarm := FALSE;
  vari.generalErrorCode := 0;
  vari.readResultCode := 0;
  IF vari.alarming THEN
    triggerStep := 0;
  END_IF;
END_IF;
errorClear := machine.reset;

IF NOT vari.disabled THEN
  //一般错误报警
  IF error
    OR generalErrorCode <> 0
  THEN
    vari.generalError := TRUE;
    vari.generalErrorCode :=generalErrorCode;
  END_IF;
  
  // //读取错误报警
  // IF failure.readFailure
  //   OR resultCode.readResultCode <> 0
  // THEN
  //   vari.readError := TRUE;
  //   vari.readResultCode := resultCode.readResultCode;
  // END_IF;
  
  //超时报警
  timeoutTimer(IN:= vari.busy,
  			   PT:= data.timeout);
  IF NOT vari.readTimeoutDisabled AND data.timeout > T#0MS AND timeoutTimer.Q THEN
  	vari.readTimeoutAlarm:=TRUE;
  END_IF;
END_IF;

//工站报警中
vari.alarming := vari.generalError OR vari.readError OR vari.readTimeoutAlarm;
//反馈工站报警
IF vari.alarming THEN
  machine.alarmCount := machine.alarmCount +1;
  station.report.alarming := TRUE;
END_IF;
END_ACTION

ACTION Cache:
//-----------------------------------------Cache-----------------------------------------//
  
resetCache := machine.reset;
triggerHmiCache := vari.triggerHmi;
triggerAutoCache := vari.triggerAuto;
vari.triggerAuto := FALSE;
END_ACTION

ACTION General:
//-----------------------------------------General-----------------------------------------//  
  
//准备就绪
vari.ready := NOT allbusy
AND NOT trgBusy
AND NOT vari.readError
AND NOT vari.generalError
AND NOT vari.readTimeoutAlarm;
//触发允许操作
vari.triggerAllow := machine.eStop
AND vari.ready;
//触发禁止图标
vari.triggerForbidIcon := NOT machine.manualMode OR NOT vari.triggerAllow;

//状态
IF vari.generalError THEN
  vari.status := ERR_GENERAL;
ELSIF vari.readError THEN
  vari.status := ERR_READL;
ELSIF vari.readTimeoutAlarm THEN
  vari.status := ERR_TIMEOUT;
ELSIF vari.busy THEN
  vari.status := BUSY;
ELSIF vari.done THEN
  vari.status := READ_SUCCESS;
ELSIF vari.ready THEN
  vari.status := READY;
ELSE
  vari.status := 0;
END_IF;
END_ACTION

ACTION InPutUpdate:
//-----------------------------------------InPutUpdate-----------------------------------------//
  
  // 输入更新
error					:= vari.input[0].0;
readComplete			:= vari.input[1].0;
generalErrorCode		:= WORD_TO_UINT(vari.input[16]);
resultDataSize			:= WORD_TO_UINT(vari.input[21]);
	
resultData[0] := WORD_TO_BYTE(SHR(vari.input[22], 8));
resultData[1] := WORD_TO_BYTE(vari.input[22]);

IF moduleType = N_L21 OR moduleType = SR_1000X OR moduleType = SR_2000X THEN
	allbusy				:= vari.input[0].8;
	trgBusy				:= vari.input[0].9;
END_IF;

  IF moduleType = SR_1000X OR moduleType = SR_2000X THEN
	ISO_IEC15415Grade			:=WORD_TO_UINT(vari.input[5]);
	ISO_IEC_TR29158Grade	:=WORD_TO_UINT(vari.input[6]);
  END_IF;
END_ACTION

ACTION ManualTip:
//-----------------------------------------ManualTip-----------------------------------------//
  
//整机手动提示           
IF vari.triggerHmi THEN
  machine.presetManualTips[0] := NOT machine.eStop;     //急停中,无法操作
  machine.presetManualTips[4] := NOT machine.manualMode;//不在手动模式,无法操作
END_IF;
END_ACTION

ACTION OutPutUpdate:
//-----------------------------------------OutPutUpdate-----------------------------------------//
  
// 输出更新
vari.output[0].7:=errorClear;
vari.output[0].8:=readRequest;
vari.output[1].0:=readCompleteClear;
END_ACTION

ACTION ScanFlow:
//-----------------------------------------ScanFlow-----------------------------------------//
  
//================================================================================== 
// 读取OK时 
// ...1 将“Read request”设为ON（1）。
// ...2 将“Read request”设为ON（1）时, SR-1000系列将开始读取, “TRG BUSY”变为ON（1）。
// ...3 读取条码时, 将在“Result Data”中写入数据。此时, “TRG BUSY”变为OFF（0）, “Read Complete”变为ON（1）。
// ...4 将“Read request”设为OFF（0）。
// ...5 确认“Read Complete”为ON（1）后, 将“Read Comlplete Clear”设为ON（1）。
// ...6 将“Read Comlplete Clear”设为ON（1）时, “Read Complete”变为OFF（0）。
// ...7 确认“Read Complete”为OFF（0）后, 将“Read Comlplete Clear”设为OFF（0）。
// 读取错误时
// ...1 将“Read request”设为ON（1）。
// ...2 将“Read request”设为ON（1）时, SR-1000系列将开始读取, “TRG BUSY”变为ON（1）。
// ...3 经过“单脉冲触发持续时间”后, 结束读取。
// ...4 无法读取条码, 因此将在“Result Data”中写入“错误”。将在“Read Result Code”中写入“201”。此时, “TRG BUSY”变为OFF（0）, “Read Complete”变为ON（1）。
// ...5 确认“Read Complete”为ON（1）后, 将“Read Comlplete Clear”设为ON（1）。
// ...6 将“Read Comlplete Clear”设为ON（1）时, “Read Complete”和“Read Failure”变为OFF（0）。
// ...7 确认“Read Complete”为OFF（0）后, 将“Read Comlplete Clear”设为OFF（0）。
//================================================================================== 

IF NOT machine.eStop THEN
  triggerStep := 0;
END_IF;

CASE triggerStep OF
    
  0://Home triggerStep
    readRequest := FALSE;
    readCompleteClear := FALSE;
    vari.busy := FALSE;
    IF vari.triggerAllow
      AND (NOT triggerAutoCache AND vari.triggerAuto  //自动触发上升沿
      OR triggerHmiCache AND NOT vari.triggerHmi AND machine.manualMode)//手动触发下降沿
    THEN
      vari.scanGrade := LEVEL_INVALID;
      vari.resultData := '';
      vari.result := 0;
      vari.done := FALSE;
      vari.busy := TRUE;
      IF readComplete THEN
        triggerStep := triggerStep + 5;
      ELSE
        triggerStep := triggerStep + 10;
      END_IF;
    END_IF;
    
  5://读取完成清除
    readCompleteClear := TRUE;
    IF NOT readComplete THEN
      readCompleteClear := FALSE;
      triggerStep := triggerStep + 5;
    END_IF;
    
  10://扫码读取请求
    readRequest := TRUE;
    IF trgBusy
      OR readComplete
      OR isTimeoutTimer
    THEN
      triggerStep := triggerStep + 10;
    END_IF;
    
  20://扫码中，等待读取完成
    IF NOT trgBusy
      AND readComplete
      OR isTimeoutTimer
    THEN
      triggerStep := triggerStep + 10;
    ELSIF isTimeoutTimer OR vari.disabled THEN
      triggerStep := 50;
    END_IF;
    
  30://读取数据
	IF resultDataSize > 0 THEN
		FOR index := 0 TO MIN( resultDataSize, UINT#128)
		DO
			vari.resultData:= CONCAT(vari.resultData,BYTE_TO_STRING(resultData[index]));
		END_FOR
	END_IF;
	IF moduleType = SR_1000X OR moduleType = SR_2000X THEN
		triggerStep := triggerStep + 10;//只有在SR-1000和SR-2000型号有读取码的等级
	ELSE
		triggerStep := 50;
	END_IF;
    
  40://读取评估等级
	IF data.evaluationMode = ISO_IEC_15415 THEN    //使用ISO/IEC 15415标准
		vari.scanGrade := ISO_IEC15415Grade;
	ELSIF data.evaluationMode = ISO_IEC_TR_29158 THEN  //使用ISO/IEC TR 29158标准
		vari.scanGrade := ISO_IEC_TR29158Grade;
	ELSIF data.evaluationMode = ISO_IEC_16022 THEN  //使用ISO/IEC 16022标准
		gradeCache := BYTE_TO_INT(resultData[resultDataSize - 2]);
		CASE gradeCache OF
			65:
				vari.scanGrade := LEVEL_A;
			66:
				vari.scanGrade := LEVEL_B;
			67:
				vari.scanGrade := LEVEL_C;
			68:
				vari.scanGrade := LEVEL_D;
			70:
				vari.scanGrade := LEVEL_F;
		ELSE
			vari.scanGrade := LEVEL_INVALID;
		END_CASE;
	END_IF;
	triggerStep := triggerStep + 10;
    
  50://复位读取请求
    readRequest := FALSE;
    IF NOT readRequest THEN
      triggerStep := triggerStep + 10;
    END_IF;
    
  60://读取完成清除
    readCompleteClear := TRUE;
    IF NOT readComplete
      OR isTimeoutTimer
    THEN
      triggerStep := triggerStep + 10;
    END_IF;
    
  70://读取完成清除复位
    readCompleteClear := FALSE;
    IF NOT readCompleteClear THEN
      triggerStep := triggerStep + 10;
    END_IF;
    
  80://结果处理
    IF vari.scanGrade >= data.evaluationGrade
      AND vari.scanGrade <= LEVEL_A
      OR data.evaluationMode = 0
      OR vari.disabled
    THEN
      vari.result := RESULT_PASS;
    ELSIF isTimeoutTimer THEN
      vari.result := RESULT_TIMEOUT;
    ELSE
      vari.result := RESULT_FAIL;
    END_IF;
    triggerStep := 999;
    
  999://读取完成 
    vari.busy := FALSE;
    vari.done := TRUE;
    triggerStep := 0;
    
END_CASE;
END_ACTION

ACTION SetUp:
//-----------------------------------------SetUp-----------------------------------------//
  
IF NOT activated THEN
  activated:=TRUE;
  // 判断型号
  IF vari.sensorSeries = 'N-L20' THEN
    moduleType := N_L21;
  ELSIF vari.sensorSeries = 'SR-1000X' THEN
    moduleType := SR_1000X;
  ELSIF vari.sensorSeries = 'SR-2000X' THEN
    moduleType := SR_2000X;
  ELSIF vari.sensorSeries = 'SR-LR1' THEN
    moduleType := SR_LR1;
  END_IF;
  vari.subDisplay.2:=moduleType = SR_1000X OR moduleType = SR_2000X;
END_IF;
END_ACTION

END_FUNCTION_BLOCK

// ---- Standard/Module/Connector/Termininal/FB_Terminal_RD.TcPOU
FUNCTION_BLOCK FB_Terminal_RD
VAR_IN_OUT
machine : UDT_Machine_RD; //
station : UDT_Station_RD; //
vari : UDT_TerminalVar_RD; //
data : UDT_TerminalData_RD; //
axis : ARRAY[*] OF  UDT_AxisVar_RD; //
END_VAR
VAR_OUTPUT
END_VAR
VAR
terminalSensor : FB_Sensor_RD; //
coverSensor : FB_Sensor_RD; //
pinSensor : FB_Sensor_RD; //
safetyPermit : BOOL; //安全条件
hmiCache : BOOL; //
autoCache : BOOL; //
isTimeout : BOOL; //
camInHomePos : BOOL; //插针凸轮轴在原点位置
camNo : UINT; //
sendNo : UINT; //
timeoutTimer : TON; //超时 
activat : BOOL; //
TerminalAlarmDelay : TON; //
CoverAlarmDelay : TON; //
END_VAR

VAR CONSTANT
HOME 	     : UINT :=1 ; // 原点位置
FEED 		 : UINT :=2 ; // 送端子位置
RETREAT    	 : UINT :=3 ; // 退端子位置
PRE      	 : UINT :=4 ; // 预送端子
CIRCLE       : UINT :=2 ; // 转一圈位置
STATUS_ALARM : UINT :=1 ; // 状态Alarm
STATUS_BUSY  : UINT :=2 ; // 状态Busy
STATUS_READY : UINT :=3 ; // 状态Ready
END_VAR

SetUp();
Alarm();
General();

ACTION Alarm:
//---------------------------------------Alarm-------------------------------------------------------//
 //报警
IF	machine.reset THEN
	vari.timeoutAlarm:=FALSE;
	vari.lackTerminalAlarm:=FALSE;
	vari.CoverAlarm:=FALSE;
END_IF;

//对端子超时报警
timeoutTimer(IN:= vari.busy,
			 PT:= data.timeout);
IF	timeoutTimer.Q THEN ;
	vari.timeoutAlarm:=TRUE;
END_IF;

(*TerminalAlarmDelay(In:=Station.running AND NOT vari.terminalSensor.input 
								AND Station.flow[1].actStep=UINT#10 AND NOT Machine.dryRun 
								AND NOT vari.disable,PT:=T#1S);*)
CoverAlarmDelay(In:=Station.running AND NOT vari.coverSensor.input 
							AND NOT Machine.dryRun AND NOT vari.disable,PT:=T#1S);
IF Station.running AND NOT vari.terminalSensor.input 
	AND Station.flow[1].actStep=UINT#10 AND NOT Machine.dryRun 
	AND NOT vari.disable THEN 
	vari.lackTerminalAlarm:=TRUE;
END_IF;	
IF CoverAlarmDelay.Q THEN 
	vari.CoverAlarm:=TRUE;
END_IF;	

vari.alarming := vari.timeoutAlarm OR vari.lackTerminalAlarm OR vari.CoverAlarm;
//反馈报警中
IF vari.alarming THEN
	Machine.alarmCount :=machine.alarmCount+1;
   station.report.alarming := TRUE;
END_IF;
END_ACTION

ACTION General:
 //---------------------------------------General-----------------------------------------------------//
//安全条件
safetyPermit:=	machine.estop //急停
				AND machine.safety//设备安全
				AND machine.airOn //气压Ok
				AND machine.allDoorClosed;//安全门关闭
				
//对端子可动作			
vari.ready:=	safetyPermit
				AND vari.permit 	//动作条件
				AND vari.coverSensor.isOn 	//盖板在位
				AND vari.terminalSensor.isOn	//尾料感应器
				AND axis[sendNo].ready//送端子伺服就绪
				AND (axis[camNo].ready OR NOT vari.camAxisEnable);//插针凸轮轴准备就绪
				
vari.forbidIcon:= NOT vari.ready OR NOT machine.manualMode;				
camInHomePos:=axis[camNo].inPos[HOME] OR NOT vari.camAxisEnable;



//----------------------------------------------------------------------------------------------------//
vari.manual:=	(hmiCache AND NOT vari.hmi)    //HMI下降沿
					AND machine.manualMode //手动模式
					AND vari.ready;//对端子可动作
					
//vari.auto:=machine.start        //设备启动
//				AND machine.autoMode //自动模式
//				AND vari.ready//对端子可动作
//				AND machine.initDone //设备初始化完成
//				AND NOT vari.done//对端子未完成
//				AND NOT vari.busy//不在对端子中
//				AND NOT machine.dryRun //设备不在空跑中
//				AND NOT station.alarming; //工站不在报警中

IF	axis[sendNo].jogBackwardsHmi//送端子轴jog
	OR axis[sendNo].jogForwardHmi//送端子轴jog
	OR (axis[sendNo].moveHmi AND (axis[sendNo].movehmiNo = FEED OR axis[sendNo].movehmiNo = RETREAT)) 
	OR station.initing 
	//OR  NOT vari.permit
	OR vari.alarming
THEN
	vari.busy:=FALSE;
	vari.done:=FALSE;	//复位对端子完成信号
ELSIF vari.manual  
	OR (NOT autoCache AND vari.auto) AND  camInHomePos//插针凸轮轴在原点位置
THEN
	vari.busy:=TRUE;//对端子中
END_IF;


IF vari.busy THEN
	CASE vari.flowStep OF
 		0://流程首步
				vari.done:=FALSE;
				vari.flowStep:=vari.flowStep+1;
				
 		1://送端子原点
			IF  axis[sendNo].inPos[HOME] THEN
				vari.flowStep:=vari.flowStep+1;
			ELSE
				axis[sendNo].moveAutoNo:=HOME;
			END_IF;
			
 		2://端子检测
 			IF vari.pinSensor.isOn THEN
				vari.flowStep:=3;
			ELSIF vari.pinSensor.isOff THEN
				vari.flowStep:=5;
			END_IF;
			
 		3://退端子
 			axis[sendNo].moveAutoNo:=RETREAT;
			IF axis[sendNo].busy THEN
				vari.flowStep:=vari.flowStep+1;
			END_IF;
			
 		4://等待退端子
 			IF 	NOT axis[sendNo].busy 
				AND  axis[sendNo].inPos[HOME]
			THEN
				vari.flowStep:=2;
			END_IF;

 		5://进端子
		 	axis[sendNo].moveAutoNo:=FEED;
			IF axis[sendNo].busy THEN
				vari.flowStep:=vari.flowStep+1;
			END_IF;
			
  		6://等待进端子
			IF 	NOT axis[sendNo].Busy 
				AND  axis[sendNo].inPos[HOME]
			THEN
				vari.flowStep:=vari.flowStep+1;
			END_IF;
			
  		7://端子检测
		 	IF vari.pinSensor.isOn THEN
				vari.flowStep:=8;
			ELSIF vari.pinSensor.isOff THEN
				vari.flowStep:=5;
			END_IF;
			
		8://预送端子
 			axis[sendNo].moveAutoNo:=PRE;
			IF axis[sendNo].busy THEN
				vari.flowStep:=vari.flowStep+1;
			END_IF;
			
  		9://等待送端子轴到位
			IF 	NOT axis[sendNo].busy 
				AND  axis[sendNo].inPos[HOME]
				AND NOT axis[sendNo].error
			THEN
				IF vari.camAxisEnable AND vari.cutEnable THEN
					vari.flowStep:=10;
				ELSE
					vari.flowStep:=12;
				END_IF;
			END_IF;
			
 		10://裁切动作
 			axis[camNo].moveAutoNo:=CIRCLE;
			IF axis[camNo].busy THEN
				vari.flowStep:=vari.flowStep+1;
			END_IF;
			
 		11://等待裁切动作
 			IF	NOT axis[camNo].busy  
				AND axis[camNo].inPos[HOME]
			THEN
 				vari.flowStep:=12;
			END_IF;

 		12://对端子完成
 			vari.done:=TRUE;
			vari.flowStep:=0;
		    vari.busy:=FALSE;

	END_CASE;
ELSE
	vari.flowStep:=0;
END_IF;

  //状态
  IF vari.alarming THEN
    vari.status := STATUS_ALARM;
  ELSIF vari.busy THEN
    vari.status := STATUS_BUSY;
  ELSIF vari.ready THEN
    vari.status := STATUS_READY;
  ELSE
    vari.status := 0;
  END_IF;

hmiCache :=vari.hmi;
autoCache :=vari.auto;
vari.auto:=FALSE;
END_ACTION

ACTION SetUp:
//-----------------------------------------SetUp-----------------------------------------//
  
IF NOT activat THEN
  activat:=TRUE;
  // 判断型号
  vari.permit:=TRUE;
END_IF;

terminalSensor(machine:=machine,
			   station:=station,
			   vari:=vari.terminalSensor,
			   data:=data.terminalSensor
			   );
coverSensor(machine:=machine,
			station:=station,
			vari:=vari.coverSensor,
			data:=data.coverSensor
			);
pinSensor(machine:=machine,
		  station:=station,
		  vari:=vari.pinSensor,
		  data:=data.pinSensor
		  );
camNo:=vari.camAxisNo;
sendNo:=vari.sendAxisNo;
END_ACTION

END_FUNCTION_BLOCK

// ---- Standard/Unit/13 Valve/FB_Valve_RD.TcPOU
FUNCTION_BLOCK FB_Valve_RD
VAR_IN_OUT
machine : UDT_Machine_RD; //
station : UDT_Station_RD; //
vari : UDT_ValveVar_RD; //
data : UDT_ValveData_RD; //
END_VAR
VAR_OUTPUT
END_VAR
VAR
safetyPermit : BOOL; // 安全条件
hmiCache : Bool; // Hmi缓存
holdTimer : TON; // 延时器
activated : Bool; // 块已运行

END_VAR

//单电磁阀控制
SetUp();
General();
Manual();
AutoTip();
ManualTip();
Output();

ACTION AutoTip:
//-------------------------------------------------AutoTip-------------------------------------------------//
  
//自动提示
vari.autoTip := vari.manual;

//反馈工站自动提示
IF vari.autoTip THEN
  station.report.autoTip := TRUE;
END_IF;
END_ACTION

ACTION General:
//-------------------------------------------------General-------------------------------------------------//
  
//安全条件
safetyPermit := machine.eStop
AND machine.safety
AND machine.airOn
AND machine.allDoorClosed;
//允许阀操作
vari.allow := safetyPermit AND vari.permit;
//禁止图标
vari.forbidIcon := NOT machine.manualMode OR NOT vari.allow;
END_ACTION

ACTION Manual:
//-------------------------------------------------Manual-------------------------------------------------//
  
//手动操作
IF machine.manualMode AND vari.allow THEN
  IF hmiCache AND NOT vari.hmi THEN
    vari.manual := NOT vari.manual;
  END_IF;
END_IF;
hmiCache := vari.hmi;
END_ACTION

ACTION ManualTip:
//-------------------------------------------------ManualTip-------------------------------------------------//
  
//复位手动提示
IF machine.tipReset THEN
  vari.manualTip := FALSE;
END_IF;

//手动提示           
IF vari.hmi THEN
  machine.presetManualTips[0] := NOT machine.eStop;     //急停中,无法操作
  machine.presetManualTips[1] := NOT machine.safety;    //安全条件不满足,无法操作
  machine.presetManualTips[2] := NOT machine.allDoorClosed;  //安全门未锁好,无法操作
  machine.presetManualTips[3] := NOT machine.airOn;     //气压不足,无法操作
  machine.presetManualTips[4] := NOT machine.manualMode;//不在手动模式,无法操作
  IF safetyPermit AND NOT vari.permit THEN
    vari.manualTip := TRUE;  //条件不满足，无法操作
  END_IF;
END_IF;

//反馈工站手动提示
IF vari.manualTip THEN
  station.report.manualTip := TRUE;
END_IF;
END_ACTION

ACTION Output:
//-------------------------------------------------Output-------------------------------------------------//
  
//急停和初始化时复位手动/自动执行
IF vari.init OR NOT machine.eStop THEN
  vari.manual := FALSE;
  vari.auto := FALSE;
END_IF;

//阀输出
vari.valve := safetyPermit AND (vari.manual XOR vari.auto);

//阀输出延时
holdTimer(IN := vari.valve,
           PT := data.holdTime,
           Q => vari.isOn);

IF data.holdTime > T#0MS AND vari.isOn THEN
  vari.auto := FALSE;
  vari.manual := FALSE;
END_IF;
END_ACTION

ACTION SetUp:
//-------------------------------------------------SetUp-------------------------------------------------//
  
IF NOT activated THEN
  activated:=TRUE;
  vari.stationNo:=0;
  // 初始值赋值
vari.permit:=TRUE;
END_IF;
END_ACTION

END_FUNCTION_BLOCK

// ---- Standard/Public/00 System/FB_GetPlcClock.TcPOU
FUNCTION_BLOCK FB_GetPlcClock


VAR_IN_OUT 
clock :  UDT_Clock_RD;
END_VAR

VAR 
fbBlinker : ARRAY[1..6] OF FB_Blinker_RD; 
END_VAR

ACT();

ACTION ACT:
fbBlinker[1](
	OnTime:= T#1MS, 
	OffTime:= T#1MS, 
	clock=> clock.c1ms, 
	R_Plus=> clock.p1ms, 
	F_Plus=> );

fbBlinker[2](
	OnTime:= T#10MS, 
	OffTime:= T#10MS, 
	clock=> clock.c10ms, 
	R_Plus=> clock.p10ms, 
	F_Plus=> );

fbBlinker[3](
	OnTime:= T#20MS, 
	OffTime:= T#20MS, 
	clock=> clock.c20ms, 
	R_Plus=> clock.p20ms, 
	F_Plus=> );
  
  
fbBlinker[4](
	OnTime:= T#100MS, 
	OffTime:= T#100MS, 
	clock=> clock.c100ms, 
	R_Plus=> clock.p100ms, 
	F_Plus=> );


fbBlinker[5](
	OnTime:= T#1000MS, 
	OffTime:= T#1000MS, 
	clock=> clock.c1s, 
	R_Plus=> clock.p1s, 
	F_Plus=> );
  
  
fbBlinker[6](
	OnTime:= T#1M, 
	OffTime:= T#1M, 
	clock=> clock.c1min, 
	R_Plus=> clock.p1min, 
	F_Plus=> );
END_ACTION

END_FUNCTION_BLOCK

// ---- Standard/Public/00 System/FB_Blinker_RD.TcPOU
FUNCTION_BLOCK FB_Blinker_RD
VAR_INPUT
	OnTime							: TIME;					//On时长
	OffTime				   		: TIME;					//Off时长
END_VAR

VAR_OUTPUT
	clock							: BOOL;					//
	R_Plus						: BOOL;					//脉冲上升沿
	F_Plus						: BOOL;					//脉冲下降沿
END_VAR

VAR
	{attribute 'hide'}
	tonOff						: TON;					//Off计时器
	{attribute 'hide'}
	tonOn						: TON;					//On计时器
END_VAR

tonOff(IN:=NOT clock, PT:=OffTime, Q=>R_Plus );
tonOn(IN:=clock, PT:=OnTime, Q=>F_Plus );

IF R_Plus OR F_Plus THEN
	clock:= NOT clock;
END_IF

END_FUNCTION_BLOCK

// ---- CheckBounds.TcPOU
// 隐含生成代码：不要编辑
FUNCTION CheckBounds : DINT
VAR_INPUT
	index, lower, upper: DINT;
END_VAR

// 隐含生成代码：这里只是对代码实现的建议
{noflow}
IF  index < lower THEN
	CheckBounds := lower;
ELSIF  index > upper THEN
	CheckBounds := upper;
ELSE  
	CheckBounds := index;
END_IF
{flow}

END_FUNCTION

// ---- CheckDivDInt.TcPOU
// 隐含生成代码：不要编辑
FUNCTION CheckDivDInt : DINT
VAR_INPUT
	divisor:DINT;
END_VAR

// 隐含生成代码：这里只是对代码实现的建议
{noflow}
IF divisor = 0 THEN
	CheckDivDInt:=1;
ELSE
	CheckDivDInt:=divisor;
END_IF;
{flow}

END_FUNCTION

// ---- CheckDivLInt.TcPOU
// 隐含生成代码：不要编辑
FUNCTION CheckDivLInt : LINT
VAR_INPUT
	divisor:LINT;
END_VAR

// 隐含生成代码：这里只是对代码实现的建议
{noflow}
IF divisor = 0 THEN
	CheckDivLInt:=1;
ELSE
	CheckDivLInt:=divisor;
END_IF;
{flow}

END_FUNCTION

// ---- CheckDivLReal.TcPOU
// 隐含生成代码：不要编辑
FUNCTION CheckDivLReal : LREAL
VAR_INPUT
	divisor:LREAL;
END_VAR

// 隐含生成代码：这里只是对代码实现的建议
{noflow}
IF divisor = 0 THEN
	CheckDivLReal:=1;
ELSE
	CheckDivLReal:=divisor;
END_IF;
{flow}

END_FUNCTION

// ---- CheckDivReal.TcPOU
// 隐含生成代码：不要编辑
FUNCTION CheckDivReal : REAL
VAR_INPUT
	divisor:REAL;
END_VAR

// 隐含生成代码：这里只是对代码实现的建议
{noflow}
IF divisor = 0 THEN
	CheckDivReal:=1;
ELSE
	CheckDivReal:=divisor;
END_IF;
{flow}

END_FUNCTION

// ---- CheckLRangeSigned.TcPOU
// 隐含生成代码：不要编辑
FUNCTION CheckLRangeSigned : LINT
VAR_INPUT
	value, lower, upper: LINT;
END_VAR

// 隐含生成代码：这里只是对代码实现的建议
{noflow}
IF (value < lower) THEN
	CheckLRangeSigned := lower;
ELSIF(value > upper) THEN
	CheckLRangeSigned := upper;
ELSE
	CheckLRangeSigned := value;
END_IF

{flow}

END_FUNCTION

// ---- CheckLRangeUnsigned.TcPOU
// 隐含生成代码：不要编辑
FUNCTION CheckLRangeUnsigned : ULINT
VAR_INPUT
	value, lower, upper: ULINT;
END_VAR

// 隐含生成代码：这里只是对代码实现的建议
{noflow}
IF (value < lower) THEN
	CheckLRangeUnsigned := lower;
ELSIF(value > upper) THEN
	CheckLRangeUnsigned := upper;
ELSE
	CheckLRangeUnsigned := value;
END_IF
{flow}

END_FUNCTION

// ---- CheckPointer.TcPOU
// 隐含生成代码：不要编辑
FUNCTION CheckPointer : POINTER TO BYTE
VAR_INPUT 
	ptToTest : POINTER TO BYTE; // 指针的目标地址
	iSize : DINT;		        // 指针指向的类型大小。（例如：POINTER TO ARRAY [0..9] OF INT为20）
	iGran : DINT;		        // 指针访问的粒度，即指针指向的类型中最大的非结构数据类型的大小。（例如：POINTER TO ARRAY [0..9] OF INT为2）
	bWrite: BOOL;		        // 指示读或写权限。TRUE=写权限。
END_VAR

// 隐含生成代码：这里只是对代码实现的建议
{noflow}
IF ptToTest=0 THEN
    ADSLOGSTR(ADSLOG_MSGTYPE_ERROR OR ADSLOG_MSGTYPE_STRING,'CheckPointer failed due to invalid address.','');
ELSIF iSize<=0 THEN
    ADSLOGSTR(ADSLOG_MSGTYPE_ERROR OR ADSLOG_MSGTYPE_STRING,'CheckPointer failed due to invalid size.','');
ELSIF iGran<=0 THEN
    ADSLOGSTR(ADSLOG_MSGTYPE_ERROR OR ADSLOG_MSGTYPE_STRING,'CheckPointer failed due to invalid granularity.','');
// -> Please note that the following memory area check is time consuming:
//ELSIF F_CheckMemoryArea(pData:=ptToTest,nSize:=DINT_TO_UDINT(iSize)) = E_TcMemoryArea.Unknown THEN
//    ADSLOGSTR(ADSLOG_MSGTYPE_ERROR OR ADSLOG_MSGTYPE_STRING,'CheckPointer failed due to unknown memory area.','');
END_IF
CheckPointer := ptToTest;
{flow}

END_FUNCTION

// ---- CheckRangeSigned.TcPOU
// 隐含生成代码：不要编辑
FUNCTION CheckRangeSigned : DINT
VAR_INPUT
	value, lower, upper: DINT;
END_VAR

// 隐含生成代码：这里只是对代码实现的建议
{noflow}
IF (value < lower) THEN
	CheckRangeSigned := lower;
ELSIF(value > upper) THEN
	CheckRangeSigned := upper;
ELSE
	CheckRangeSigned := value;
END_IF
{flow}

END_FUNCTION

// ---- CheckRangeUnsigned.TcPOU
// 隐含生成代码：不要编辑
FUNCTION CheckRangeUnsigned : UDINT
VAR_INPUT
	value, lower, upper: UDINT;
END_VAR

// 隐含生成代码：这里只是对代码实现的建议
{noflow}
IF (value < lower) THEN
	CheckRangeUnsigned := lower;
ELSIF(value > upper) THEN
	CheckRangeUnsigned := upper;
ELSE
	CheckRangeUnsigned := value;
END_IF
{flow}

END_FUNCTION

// ---- Standard/FUN/FUN_WordToAry.TcPOU
FUNCTION FUN_WordToAry : ARRAY[0..15] OF BOOL
VAR_INPUT
	in : WORD;
END_VAR
VAR
END_VAR

FUN_WordToAry[0]:=in.0;
FUN_WordToAry[1]:=in.1;
FUN_WordToAry[2]:=in.2;
FUN_WordToAry[3]:=in.3;
FUN_WordToAry[4]:=in.4;
FUN_WordToAry[5]:=in.5;
FUN_WordToAry[6]:=in.6;
FUN_WordToAry[7]:=in.7;
FUN_WordToAry[8]:=in.8;
FUN_WordToAry[9]:=in.9;
FUN_WordToAry[10]:=in.10;
FUN_WordToAry[11]:=in.11;
FUN_WordToAry[12]:=in.12;
FUN_WordToAry[13]:=in.13;
FUN_WordToAry[14]:=in.14;
FUN_WordToAry[15]:=in.15;

END_FUNCTION

// ---- Standard/FUN/F_Sum.TcPOU
FUNCTION F_Sum : DINT;
VAR_IN_OUT
    aData     : ARRAY [*] OF DINT;
END_VAR
VAR
    i, nSum   : DINT;
END_VAR


nSum := 0;
FOR i := LOWER_BOUND(aData,1) TO UPPER_BOUND(aData,1) DO
    nSum := nSum + aData[i];
END_FOR;
F_Sum := nSum;

END_FUNCTION

// ---- Standard/Module/Connector/Termininal/FB_Terminal2_RD.TcPOU
FUNCTION_BLOCK FB_Terminal2_RD
VAR_IN_OUT
machine : UDT_Machine_RD; //
station : UDT_Station_RD; //
vari : UDT_TerminalVar_RD; //
data : UDT_TerminalData_RD; //
axis : ARRAY[*] OF  UDT_AxisVar_RD; //
END_VAR
VAR_OUTPUT
END_VAR
VAR
terminalSensor : FB_Sensor_RD; //
coverSensor : FB_Sensor_RD; //
pinSensor : FB_Sensor_RD; //
safetyPermit : BOOL; //安全条件
hmiCache : BOOL; //
autoCache : BOOL; //
isTimeout : BOOL; //
camInHomePos : BOOL; //插针凸轮轴在原点位置
camNo : INT; //
sendNo : INT; //
timeoutTimer : TON; //超时 
activat : BOOL; //
TerminalAlarmDelay : TON; //
CoverAlarmDelay : TON; //
END_VAR

VAR CONSTANT
HOME 	     : INT :=1 ; // 原点位置
FEED 		 : INT :=2 ; // 送端子位置
RETREAT    	 : INT :=3 ; // 退端子位置
PRE      	 : INT :=4 ; // 预送端子
CIRCLE       : INT :=2 ; // 转一圈位置
STATUS_ALARM : INT :=1 ; // 状态Alarm
STATUS_BUSY  : INT :=2 ; // 状态Busy
STATUS_READY : INT :=3 ; // 状态Ready
END_VAR

SetUp();
Alarm();
General();

ACTION Alarm:
//---------------------------------------Alarm-------------------------------------------------------//
 //报警
IF	machine.reset THEN
	vari.timeoutAlarm:=FALSE;
	vari.lackTerminalAlarm:=FALSE;
	vari.CoverAlarm:=FALSE;
END_IF;

//对端子超时报警
timeoutTimer(IN:= vari.busy,
			 PT:= data.timeout);
IF	timeoutTimer.Q THEN ;
	vari.timeoutAlarm:=TRUE;
END_IF;

(*TerminalAlarmDelay(In:=Station.running AND NOT vari.terminalSensor.input 
								AND Station.flow[1].actStep=UINT#10 AND NOT Machine.dryRun 
								AND NOT vari.disable,PT:=T#1S);*)
CoverAlarmDelay(In:=Station.running AND NOT vari.coverSensor.input 
							AND NOT Machine.dryRun AND NOT vari.disable,PT:=T#1S);
IF Station.running AND NOT vari.terminalSensor.input 
	AND Station.flow[1].actStep=UINT#10 AND NOT Machine.dryRun 
	AND NOT vari.disable THEN 
	vari.lackTerminalAlarm:=TRUE;
END_IF;	
IF CoverAlarmDelay.Q THEN 
	vari.CoverAlarm:=TRUE;
END_IF;	

vari.alarming := vari.timeoutAlarm OR vari.lackTerminalAlarm OR vari.CoverAlarm;
//反馈报警中
IF vari.alarming THEN
	Machine.alarmCount :=machine.alarmCount+1;
   station.report.alarming := TRUE;
END_IF;
END_ACTION

ACTION General:
 //---------------------------------------General-----------------------------------------------------//
//安全条件
safetyPermit:=	machine.estop //急停
				AND machine.safety//设备安全
				AND machine.airOn //气压Ok
				AND machine.allDoorClosed;//安全门关闭
				
//对端子可动作			
vari.ready:=	safetyPermit
				AND vari.permit 	//动作条件
				AND vari.coverSensor.isOn 	//盖板在位
				AND vari.terminalSensor.isOn	//尾料感应器
				AND axis[sendNo].ready//送端子伺服就绪
				AND (axis[camNo].ready OR NOT vari.camAxisEnable);//插针凸轮轴准备就绪
				
vari.forbidIcon:= NOT vari.ready OR NOT machine.manualMode;				
camInHomePos:=axis[camNo].inPos[HOME] OR NOT vari.camAxisEnable;



//----------------------------------------------------------------------------------------------------//
vari.manual:=	(hmiCache AND NOT vari.hmi)    //HMI下降沿
					AND machine.manualMode //手动模式
					AND vari.ready;//对端子可动作
					
//vari.auto:=machine.start        //设备启动
//				AND machine.autoMode //自动模式
//				AND vari.ready//对端子可动作
//				AND machine.initDone //设备初始化完成
//				AND NOT vari.done//对端子未完成
//				AND NOT vari.busy//不在对端子中
//				AND NOT machine.dryRun //设备不在空跑中
//				AND NOT station.alarming; //工站不在报警中

IF	axis[sendNo].jogBackwardsHmi//送端子轴jog
	OR axis[sendNo].jogForwardHmi//送端子轴jog
	OR (axis[sendNo].moveHmi AND (axis[sendNo].movehmiNo = FEED OR axis[sendNo].movehmiNo = RETREAT)) 
	OR station.initing 
	//OR  NOT vari.permit
	OR vari.alarming
THEN
	vari.busy:=FALSE;
	vari.done:=FALSE;	//复位对端子完成信号
ELSIF vari.manual  
	OR (NOT autoCache AND vari.auto) AND  camInHomePos//插针凸轮轴在原点位置
THEN
	vari.busy:=TRUE;//对端子中
END_IF;


IF vari.busy THEN
	CASE vari.flowStep OF
 		0://流程首步
				vari.done:=FALSE;
				vari.flowStep:=vari.flowStep+1;
				
 		1://送端子原点
			IF  axis[sendNo].inPos[HOME] THEN
				vari.flowStep:=vari.flowStep+1;
			ELSE
				axis[sendNo].moveAutoNo:=HOME;
			END_IF;
			
 		2://端子检测
 			IF vari.pinSensor.isOn THEN
				vari.flowStep:=3;
			ELSIF vari.pinSensor.isOff THEN
				vari.flowStep:=5;
			END_IF;
			
 		3://退端子
 			axis[sendNo].moveAutoNo:=RETREAT;
			IF axis[sendNo].busy THEN
				vari.flowStep:=vari.flowStep+1;
			END_IF;
			
 		4://等待退端子
 			IF 	NOT axis[sendNo].busy 
				AND  axis[sendNo].inPos[HOME]
			THEN
				vari.flowStep:=2;
			END_IF;

 		5://进端子
		 	axis[sendNo].moveAutoNo:=FEED;
			IF axis[sendNo].busy THEN
				vari.flowStep:=vari.flowStep+1;
			END_IF;
			
  		6://等待进端子
			IF 	NOT axis[sendNo].Busy 
				AND  axis[sendNo].inPos[HOME]
			THEN
				vari.flowStep:=vari.flowStep+1;
			END_IF;
			
  		7://端子检测
		 	IF vari.pinSensor.isOn THEN
				vari.flowStep:=8;
			ELSIF vari.pinSensor.isOff THEN
				vari.flowStep:=5;
			END_IF;
			
		8://预送端子
 			axis[sendNo].moveAutoNo:=PRE;
			IF axis[sendNo].busy THEN
				vari.flowStep:=vari.flowStep+1;
			END_IF;
			
  		9://等待送端子轴到位
			IF 	NOT axis[sendNo].busy 
				//AND  axis[sendNo].inPos[HOME]
				AND NOT axis[sendNo].error
			THEN
				IF vari.camAxisEnable AND vari.cutEnable THEN
					vari.flowStep:=10;
				ELSE
					vari.flowStep:=12;
				END_IF;
			END_IF;
			
 		10://裁切动作
 			axis[camNo].moveAutoNo:=CIRCLE;
			IF axis[camNo].busy THEN
				vari.flowStep:=vari.flowStep+1;
			END_IF;
			
 		11://等待裁切动作
 			IF	NOT axis[camNo].busy  
				AND axis[camNo].inPos[HOME]
			THEN
 				vari.flowStep:=12;
			END_IF;

		12://进端子
		 	axis[sendNo].moveAutoNo:=FEED;
			IF axis[sendNo].busy THEN
				vari.flowStep:=vari.flowStep+1;
			END_IF;
			
  		13://等待进端子
			IF 	NOT axis[sendNo].Busy 
				AND  axis[sendNo].inPos[HOME]
			THEN
				IF vari.camAxisEnable AND vari.cutEnable THEN
					vari.flowStep:=vari.flowStep+1;
				ELSE
					vari.flowStep:=16;
				END_IF;	
			END_IF;			
			
 		14://裁切动作
 			axis[camNo].moveAutoNo:=CIRCLE;
			IF axis[camNo].busy THEN
				vari.flowStep:=vari.flowStep+1;
			END_IF;
			
 		15://等待裁切动作
 			IF	NOT axis[camNo].busy  
				AND axis[camNo].inPos[HOME]
			THEN
 				vari.flowStep:=16;
			END_IF;			

 		16://进端子
		 	axis[sendNo].moveAutoNo:=FEED;
			IF axis[sendNo].busy THEN
				vari.flowStep:=vari.flowStep+1;
			END_IF;
			
  		17://等待进端子
			IF 	NOT axis[sendNo].Busy 
				AND  axis[sendNo].inPos[HOME]
			THEN
				IF vari.camAxisEnable AND vari.cutEnable THEN
					vari.flowStep:=vari.flowStep+1;
				ELSE
					vari.flowStep:=20;
				END_IF;	
			END_IF;			
			
 		18://裁切动作
 			axis[camNo].moveAutoNo:=CIRCLE;
			IF axis[camNo].busy THEN
				vari.flowStep:=vari.flowStep+1;
			END_IF;
			
 		19://等待裁切动作
 			IF	NOT axis[camNo].busy  
				AND axis[camNo].inPos[HOME]
			THEN
 				vari.flowStep:=20;
			END_IF;	
			
 		20://对端子完成
 			vari.done:=TRUE;
			vari.flowStep:=0;
		    vari.busy:=FALSE;

	END_CASE;
ELSE
	vari.flowStep:=0;
END_IF;

  //状态
  IF vari.alarming THEN
    vari.status := STATUS_ALARM;
  ELSIF vari.busy THEN
    vari.status := STATUS_BUSY;
  ELSIF vari.ready THEN
    vari.status := STATUS_READY;
  ELSE
    vari.status := 0;
  END_IF;

hmiCache :=vari.hmi;
autoCache :=vari.auto;
vari.auto:=FALSE;
END_ACTION

ACTION SetUp:
//-----------------------------------------SetUp-----------------------------------------//
  
IF NOT activat THEN
  activat:=TRUE;
  // 判断型号
  vari.permit:=TRUE;
END_IF;

terminalSensor(machine:=machine,
			   station:=station,
			   vari:=vari.terminalSensor,
			   data:=data.terminalSensor
			   );
coverSensor(machine:=machine,
			station:=station,
			vari:=vari.coverSensor,
			data:=data.coverSensor
			);
pinSensor(machine:=machine,
		  station:=station,
		  vari:=vari.pinSensor,
		  data:=data.pinSensor
		  );
camNo:=vari.camAxisNo;
sendNo:=vari.sendAxisNo;
END_ACTION

END_FUNCTION_BLOCK

// ---- Standard/Public/03 HMI/FB_GetPageSerialNo_RD.TcPOU
FUNCTION_BLOCK FB_GetPageSerialNo_RD
VAR_IN_OUT
pageDisplayNum : INT; // 当页显示数量
maxModuleNumInStation : Int; // 单工站最大部件数
nextPage : Bool; // 下一页
prevPage : Bool; // 上一页
nextPageDisplay : Bool; // 下一页按钮显示
prevPageDisplay : Bool; // 上一页按钮显示
control : Array[0..8] of Int; // 当前工站数据
unitList : Array[*] of Int; // 当前部件显示列表

END_VAR

VAR
serialNo : DINT; // 序号
serialMax : DINT; // 最大可翻页
index : DInt; // 循环索引

END_VAR

VAR CONSTANT

PAGE_MAX_NUM : DINT := 8; // 单画面最大部件数
END_VAR

// 上下翻页
IF nextPage THEN
  serialNo := serialNo + pageDisplayNum;
ELSIF prevPage THEN
  serialNo := serialNo - pageDisplayNum;
END_IF;

// 根据当前工站部件数量和显示位置获取最大可翻页序号(例如 1,3,5,7,9)
serialMax := 0;
FOR index := maxModuleNumInStation TO 1 BY -1 DO
  IF unitList[index] <> 0 THEN
    serialMax := ((index - 1) / pageDisplayNum) * pageDisplayNum;
    EXIT;   // 获取最大位置即跳出循环
  END_IF;
END_FOR;

//清空多余页
IF pageDisplayNum < PAGE_MAX_NUM THEN
  FOR index := pageDisplayNum + 1 TO PAGE_MAX_NUM DO
    control[index] := 0;
  END_FOR;
END_IF;

// 根据最大可翻页序号,防止越界
IF serialNo > serialMax THEN
  serialNo := serialMax;
END_IF;
serialNo := LIMIT(serialNo,0,maxModuleNumInStation - pageDisplayNum);

// 显示偏移
FOR index := 1 TO pageDisplayNum DO
  IF (serialNo + index) <= maxModuleNumInStation THEN
    control[index] :=
    unitList[serialNo + index];
  ELSE
    control[index] := 0;
  END_IF;
END_FOR;

// 上/下一页显示
prevPageDisplay := serialNo > 0;
nextPageDisplay := serialNo < serialMax;

END_FUNCTION_BLOCK

// ---- Standard/Public/03 HMI/FB_GetPlcClock_RD.TcPOU
FUNCTION_BLOCK FB_GetPlcClock_RD
VAR_IN_OUT
clock         : UDT_Clock_RD;
END_VAR
VAR
c1msCache : BOOL; //
c10msCache : BOOL; //
c20msCache : BOOL; //
c100msCache : BOOL; //
c1sCache : BOOL; //
c1minCache : BOOL; //
count : DINT; //

END_VAR

PlcClock();

METHOD Blinker : BOOL
VAR_INPUT
	ltimeActive                 : BOOL;                 //激活微秒计时
	tOn							: TIME;					//On时长
	tOff						: TIME;					//Off时长
	ltOn						: LTIME;					//On时长
	ltOff						: LTIME;					//Off时长
END_VAR

VAR_OUTPUT
	bP							: BOOL;					//脉冲
	bR							: BOOL;					//脉冲上升沿
	bF							: BOOL;					//脉冲下降沿
END_VAR

VAR
	{attribute 'hide'}
	tonOff						: TON;					//Off计时器
	{attribute 'hide'}
	tonOn						: TON;					//On计时器
	{attribute 'hide'}
	ltonOff						: LTON;					//Off计时器
	{attribute 'hide'}
	ltonOn						: LTON;					//On计时器
END_VAR
IF NOT ltimeActive
THEN
	tonOff(IN:=NOT bP, PT:=tOff, Q=>bR );

    tonOn(IN:=bP, PT:=tOn, Q=>bF );
    
    IF bR OR bF THEN
    	bP:=NOT bP;
    END_IF
ELSE
	ltonOff(IN:=NOT bP, PT:=ltOff, Q=>bR );

    ltonOn(IN:=bP, PT:=ltOn, Q=>bF );
    
    IF bR OR bF THEN
    	bP:=NOT bP;
    END_IF
END_IF
END_METHOD

ACTION PlcClock:
Blinker(ltimeActive:=TRUE,tOn:=T#0MS,tOff:=T#0MS,ltOn:=LTIME#500US,ltOff:=LTIME#500US,bP=>clock.c1ms);
Blinker(ltimeActive:=FALSE,tOn:=T#5MS,tOff:=T#5MS,ltOn:=LTIME#0US,ltOff:=LTIME#0US,bP=>clock.c10ms);
Blinker(ltimeActive:=FALSE,tOn:=T#10MS,tOff:=T#10MS,ltOn:=LTIME#0US,ltOff:=LTIME#0US,bP=>clock.c20ms);
Blinker(ltimeActive:=FALSE,tOn:=T#50MS,tOff:=T#50MS,ltOn:=LTIME#0US,ltOff:=LTIME#0US,bP=>clock.c100ms);
Blinker(ltimeActive:=FALSE,tOn:=T#500MS,tOff:=T#500MS,ltOn:=LTIME#0US,ltOff:=LTIME#0US,bP=>clock.c1s);
Blinker(ltimeActive:=FALSE,tOn:=T#30S,tOff:=T#30S,ltOn:=LTIME#0US,ltOff:=LTIME#0US,bP=>clock.c1min);

clock.p1ms		:=NOT c1msCache AND clock.c1ms;
clock.p10ms		:=NOT c10msCache AND clock.c10ms;
clock.p20ms		:=NOT c20msCache	 AND clock.c20ms;
clock.p100ms	:=NOT c100msCache AND clock.c100ms;
clock.p1s			:=NOT c1sCache AND clock.c1s;
clock.p1min		:=NOT c1minCache AND clock.c1min;

IF clock.p1min THEN
  count := count +1;
  count := count MOD 60;
END_IF;
clock.p1hour	:=clock.p1min AND count = 0;

c1msCache	:=clock.c1ms;
c10msCache	:=clock.c10ms;
c20msCache	:=clock.c20ms;
c100msCache	:=clock.c100ms;
c1sCache			:=clock.c1s;
c1minCache		:=clock.c1min;
END_ACTION

END_FUNCTION_BLOCK

// ---- Standard/Public/03 HMI/FB_Hmi_RD.TcPOU
FUNCTION_BLOCK FB_Hmi_RD
VAR_INPUT
END_VAR
VAR_OUTPUT
END_VAR
VAR
END_VAR

  //================================================================================== 
  // Harmontromics / (C) Copyright (2021) 
  //----------------------------------------------------------------------------------
  // Title:               hmi
  // Comment/Function:    Operation and display of hmi interface
  // Library/Family:      (that the source is dedicated to)
  // Author:              David.Wong
  // Target System: 
  // Engineering:         Sysmac Studio
  // Restrictions:        (OB types, etc.)
  // Requirements:        (hardware, technological package, etc.) 
  //----------------------------------------------------------------------------------
  // Change log table:
  // Version     | Date       | Expert in charge | Changes applied
  //-------------|------------|------------------|------------------------------------
  // 001.000.000 | 2021-12-11 | David.Wong       | First released version
  // 001.000.001 | 2022-1-6   | David.Wong       | The multi page display of modified cylinder servo is incorrect
  // 001.000.002 | 2022-3-25  | David.Wong       | Add the lower limit detection of MAX_AXIS_IN_STATION and MAX_CYL_IN_STATION             
  // 001.001.001 | 2022-5-8   | David.Wong       | 增加传感器、扫码枪等画面的自动编号和显示
  // 001.002.000 | 2022-11-8  | David.Wong       | Unit的数量扩展为100，修复切换机器编号后无法跳转到手动/参数页面问题
  //             |            |                  | 
  //==================================================================================

END_FUNCTION_BLOCK

// ---- Standard/Public/03 HMI/FB_IV3_G120_RD.TcPOU
FUNCTION_BLOCK FB_IV3_G120_RD
VAR_IN_OUT
bEStop : BOOL; //
bShield : BOOL; //
bManualMode : BOOL; //
bAlarmReset : BOOL; //
bTriggerHmi : BOOL; //
bTriggerAuto : BOOL; //
iProgramNo : UINT; //
bChangeProgramHmi : BOOL; //
bChangeProgramAuto : BOOL; //
bOnline : BOOL; //
bReady : BOOL; //
bBusy : BOOL; //
bDone : BOOL; //
bError : BOOL; //
bTimeout : BOOL; //
bOutTrigger : BOOL; //
iCurrentProgranNo : UINT; //
nResult : UINT; //
DataLinkInput : ARRAY[0..393] OF BYTE; //
DataLinkOutput : ARRAY[0..11] OF BYTE; //

END_VAR
VAR
nIndex1 : UINT; //
nIndex2 : UINT; //
nChangeProgramStep : UINT; //
nTriggerStep : UINT; //
ftTriggerHmi : F_TRIG; //
ftChangeProgramHmi : F_TRIG; //
rtChangeProgramAuto : R_TRIG; //
rtTriggerAuto : R_TRIG; //
ftTriggerHmi_Q : BOOL; //
ftChangeProgramHmi_Q : BOOL; //
rtTriggerAuto_Q : BOOL; //
rtChangeProgramAuto_Q : BOOL; //
bChangeProgramBusy : BOOL; //
bTriggetBusy : BOOL; //
tonTimeout : TON; //
tTimeout : TIME; //
tonTimeout_Q : BOOL; //
bTriggerManual : BOOL; //
bChangProgramManual : BOOL; //
tonReady : TON; //
tReady : TIME; //
tonReady_Q : BOOL; //
InputData : ARRAY[0..29] OF BYTE; //
OutputData : ARRAY[0..5] OF BYTE; //
Data_TriggerReady : BOOL; //
Data_TriggerAck : BOOL; //
Data_Online : BOOL; //
Data_Busy : BOOL; //
Data_InspectionComplete : BOOL; //
Data_ResultValid : BOOL; //
Data_CommandFailed : BOOL; //
Data_Error : BOOL; //
Data_ProgramChangeAck : BOOL; //
Data_ResultOK : BOOL; //
Data_ResultNG : BOOL; //
Data_SoftEventAck : BOOL; //
Data_ErrorCode : INT; //
Data_CurrentProgramNo : INT; //
Data_ResultData : ARRAY[0..13] OF BYTE; //
Data_Trigger : BOOL; //
Data_ProgramChange : BOOL; //
Data_ResultAck : BOOL; //
Data_ClearError : BOOL; //
Data_ProgramNo : INT; //
bTriggerProcessDone : BOOL; //
bChangeProgramDone : BOOL; //
tonProgramNo : TON; //
bErrorChangeProgram : BOOL; //
bErrorTrigger : BOOL; //
ResultTemp : BOOL; //
fbUnpackWord   : MEM.UnpackWord;
fbUnpackDWord  : MEM.UnpackDWord;
END_VAR

Link();
Trigger();
Alarm();
Timeout();
Output();
TriggerProcess();
ChangeProgram();

ACTION Alarm:
//***********************Alarm***********************
tTimeout:=T#5S;
tonTimeout(
	IN:=bBusy,
	PT:=tTimeout,
	Q=>tonTimeout_Q);

bError:=Data_Error OR bTimeout 
			OR bErrorChangeProgram OR bErrorTrigger;

IF bAlarmReset THEN
	bTimeout:=FALSE;
	bErrorChangeProgram:=FALSE;
	bErrorTrigger:=0;
END_IF;

Data_ClearError :=bError AND bAlarmReset;
END_ACTION

ACTION ChangeProgram:
//***********************Change Program***********************
tonProgramNo(In:=nChangeProgramStep=20, PT:=T#0.1S);

CASE nChangeProgramStep OF

//start to change Program
0:	
IF bChangProgramManual		
	OR rtChangeProgramAuto_Q
THEN
	nChangeProgramStep :=nChangeProgramStep + 10;
END_IF;

//set busy
10:
	bChangeProgramDone:=FALSE;
	bChangeProgramBusy:=TRUE;
	nChangeProgramStep :=nChangeProgramStep + 10;

//set program No.
20:
	Data_ProgramNo :=iProgramNo;
IF tonProgramNo.Q THEN
	nChangeProgramStep :=nChangeProgramStep + 10;
END_IF;

//execute command
30:
	Data_ProgramChange	:=TRUE;												//execute command
IF Data_ProgramChangeAck 		//Ack 
THEN
	nChangeProgramStep :=nChangeProgramStep + 10;
END_IF;

//result
40:
	Data_ProgramChange	:=FALSE;		//execute command
IF NOT Data_ProgramChangeAck AND NOT Data_CommandFailed	//complete and not failed
THEN
	nChangeProgramStep :=nChangeProgramStep + 10;
END_IF;

IF Data_CommandFailed				//failed
THEN
	bErrorChangeProgram:=TRUE;
	nChangeProgramStep :=nChangeProgramStep + 10;
END_IF;

//
50:
	nChangeProgramStep :=nChangeProgramStep + 10;

//done
60:
	bChangeProgramDone:=TRUE;
	nChangeProgramStep :=nChangeProgramStep + 10;	

//end
70:
	IF NOT bChangeProgramHmi AND NOT bChangeProgramAuto
	THEN
		bChangeProgramDone:=FALSE;
		bChangeProgramBusy:=FALSE;
		nChangeProgramStep :=0;	
	END_IF;
	
END_CASE;
END_ACTION

ACTION Link:
//***********************Link***********************
FOR nIndex1:=0 TO 29  BY 1 DO
	InputData[nIndex1]:=DataLinkInput[nIndex1];
END_FOR;
FOR nIndex2:=0 TO 5  BY 1 DO
	DataLinkOutput[nIndex2]:=OutputData[nIndex2];
END_FOR;
//Input
	Data_TriggerAck:=InputData[0].0;						//触发响应
	Data_ProgramChangeAck:=InputData[0].0;		//程序切换响应
	Data_CommandFailed:=InputData[1].2;			//程序切换失败
	Data_ResultValid:=InputData[2].0;					//可获取结果
	Data_InspectionComplete:=InputData[2].1;		//结果更新完成，反转	
	Data_Busy:=InputData[2].2;								//Busy
	Data_Online:=InputData[2].4;							//运行
	Data_TriggerReady:=InputData[2].6;					//Ready
	Data_Error:=InputData[3].7;								//Error
	Data_ResultOK:=InputData[4].0;						//OK
	Data_ResultNG:=InputData[4].4;						//NG	
	Data_ErrorCode := WORD_TO_INT( MEM.PackBytesToWord(byHighByte:= InputData[9], byLowByte:=InputData[8] ));//报警代码
	Data_CurrentProgramNo := WORD_TO_INT( MEM.PackBytesToWord(byHighByte:= InputData[17], byLowByte:=InputData[16] ));//当前程序号

//Output	
	OutputData[0].0:=Data_Trigger;					//触发检测
	OutputData[0].2:=Data_ProgramChange;		//切换程序
	OutputData[0].3:=Data_ClearError;				//报警复位	
	OutputData[2].0:=Data_ResultAck;				//结果确认
	fbUnpackWord(
	wValue:= INT_TO_WORD(Data_ProgramNo), 
	byLowByte=> DataLinkOutput[4], 
	byHighByte=> DataLinkOutput[5], );          //程序号
END_ACTION

ACTION Output:
//***********************Output***********************
bOutTrigger:=Data_Trigger;
iCurrentProgranNo:=Data_CurrentProgramNo;

tonReady(
	IN:=NOT bBusy,
	PT:=tReady,
	Q=>tonReady_Q);

bBusy:=bChangeProgramBusy OR bTriggetBusy OR Data_Busy;
bDone:=(bTriggerProcessDone AND bTriggerAuto)
								OR (bChangeProgramDone AND bChangeProgramAuto);

bOnline:=Data_Online;
bReady:=Data_TriggerReady;
END_ACTION

ACTION Timeout:
//***********************Timeout***********************
IF tonTimeout_Q THEN
	;//bTimeout:=TRUE;
END_IF;

IF bTimeout THEN
	bBusy:=FALSE;
	Data_Trigger:=FALSE;
	Data_ProgramChange:=FALSE;
	bTriggetBusy:=FALSE;
	bChangeProgramBusy:=FALSE;
	nTriggerStep:=0;
	nChangeProgramStep:=0;
END_IF;
END_ACTION

ACTION Trigger:
//***********************Trigger ***********************
ftChangeProgramHmi(CLK:=bChangeProgramHmi AND tonReady_Q, Q=>ftChangeProgramHmi_Q );
rtChangeProgramAuto(CLK:=bChangeProgramAuto AND tonReady_Q, Q=>rtChangeProgramAuto_Q );

ftTriggerHmi(CLK:=bTriggerHmi, Q=>ftTriggerHmi_Q );
rtTriggerAuto(CLK:=bTriggerAuto AND tonReady_Q, Q=>rtTriggerAuto_Q );

bChangProgramManual:=ftChangeProgramHmi_Q
	AND bEStop
	AND bManualMode;
	
bTriggerManual:=ftTriggerHmi_Q
	AND bEStop
	AND bManualMode;
END_ACTION

ACTION TriggerProcess:
//***********************Trigger process***********************

CASE nTriggerStep OF
	
//start to trigger process
0:	
IF bTriggerManual		
	OR rtTriggerAuto_Q
THEN
	nTriggerStep :=nTriggerStep + 10;
END_IF;

//result ack
10:
	bTriggerProcessDone:=FALSE;
	nResult:=0;
	bTriggetBusy:=TRUE;
	ResultTemp:=Data_InspectionComplete;
	nTriggerStep :=nTriggerStep + 10;

//trigger
 20:
	Data_Trigger:=TRUE;
IF ResultTemp<>Data_InspectionComplete OR bShield
THEN
	nTriggerStep :=nTriggerStep + 10;
 END_IF;
 
 //reset trigger
30:
 	Data_Trigger:=FALSE;
	IF Data_ResultOK AND NOT  Data_ResultNG		//Result output,1:OK,2:=NG
	THEN
		nResult:=1;
	ELSE
		nResult:=2;
	END_IF;	
	nTriggerStep :=nTriggerStep + 10;

//done
40:
	bTriggerProcessDone:=TRUE;
	nTriggerStep :=nTriggerStep + 10;
	
//end
50:
	IF NOT bTriggerHmi AND NOT bTriggerAuto
	THEN
		bTriggerProcessDone:=FALSE;
		bTriggetBusy:=FALSE;
		nTriggerStep :=0;	
	END_IF;

END_CASE;
END_ACTION

END_FUNCTION_BLOCK

// ---- Standard/Public/03 HMI/FB_Tben_L5_4Rfid_RD.TcPOU
FUNCTION_BLOCK FB_Tben_L5_4Rfid_RD
VAR_IN_OUT
udiStartAddress : UDINT; //
uiDataLength : UINT; //
ixRead : BOOL; //
ixWrite : BOOL; //
ixReset : BOOL; //
iarbDataTx : ARRAY[0..127] OF BYTE; //
ixChannel : UINT; //
InputData : ARRAY[0..471] OF BYTE; //
OutputData : ARRAY[0..325] OF BYTE; //
xDone : BOOL; //
xBusy : BOOL; //
xError : BOOL; //
eErrorCode : WORD; //
xTP : BOOL; //
xRWHeadNotConnected : BOOL; //
xuiDataLength : UINT; //
xarbRxData : ARRAY[0..127] OF byte; //
xarbTagUID : ARRAY[0..7] OF byte; //

END_VAR
VAR
iCommandSeq : UINT; //
iCnt01 : INT; //
iCnt02 : INT; //
bExcute : BOOL; //
wError : WORD; //
tTimout : TON; //
bOldRead : BOOL; //
bOldWrite : BOOL; //
bOldTagPresent : BOOL; //
iAdress0 : UINT; //
iAdress1 : UINT; //
iAdress2 : UINT; //
iAdress3 : UINT; //
iAdress4 : UINT; //
iAdress5 : UINT; //
InputData6_In : BYTE; //
InputData86_In : BYTE; //
InputData166_In : BYTE; //
InputData246_In : BYTE; //
ResponseCode_In : UINT; //
TagPresent_In : BOOL; //
HeadNotConnected_In : BOOL; //
ReadLength_In : UINT; //
ErrorCode_In : WORD; //
CommandCode_Out : INT; //
LoopCounter_Out : USINT; //
StartAddress_Out : DWORD; //
DataLength_Out : UINT; //
Index1 : UINT; //
Index2 : UINT; //
Index3 : UINT; //
OperationType : UINT; //
LoopCounter_In : UINT; //
rR_TRIG : ARRAY[0..5] OF R_TRIG; //
fbUnpackWord   : MEM.UnpackWord;
fbUnpackDWord  : MEM.UnpackDWord;
END_VAR

//Input And Output Address Calculate
(*
Input Data:	
系统占用2字节
CH0			CH1				CH2				CH3
2-3			82-83			162-163		242-243		ResponseCode_In				//反馈代码
4				84					164				244				LooperCounter					//LooperCounter
6.0			86.0				166.0			246.0			TP,0:No Tag 1:Tag present	//标签存在
6.7			86.7				166.7			246.7			HeadNotConnected			//读取头未连接
8-9			88-89			168-169		248-249		Length									//读取长度
10-11		90-91			170-171		250-251		Error Code							//出错代码
12-13		92-93			172-173		252-253		Tag counter							//标签计数			
26-81		106-161		186-241		266-321		Read data Byte 0-55			//读取的数据

Output Data:	
系统占用2字节
CH0			CH1				CH2				CH3
2-3			82-83			162-163		242-243		CommandCode					//命令代码
6-9			86-89			166-169		246-249		Start address						//起始地址
10-11		90-91			170-171		250-251		Length									//写入长度
26-81		86-161			186-241		266-321		Write data Byte 0-55			//写入的数据
*)

IF ixChannel=0 THEN 
	ResponseCode_In := WORD_TO_UINT( MEM.PackBytesToWord(byHighByte:= InputData[3], byLowByte:=InputData[2] ));  //2-3,反馈代码
	LoopCounter_In:=BYTE_TO_UINT(InputData[4]);						//4,LooperCounter
	InputData6_In:=InputData[6];											//6
	TagPresent_In:=InputData6_In.0;									//6.0,Tag present，标签存在
	HeadNotConnected_In:=InputData6_In.7;					//6.7,HeadNotConnected，读取头未连接
	ReadLength_In := WORD_TO_UINT( MEM.PackBytesToWord(byHighByte:= InputData[9], byLowByte:=InputData[8] ));  //ReadLength,8-9，读取到的长度
	ErrorCode_In := MEM.PackBytesToWord(byHighByte:= InputData[11], byLowByte:=InputData[10] );  //Error Code 10-11，出错代码
ELSIF ixChannel=1 THEN 
	ResponseCode_In := WORD_TO_UINT( MEM.PackBytesToWord(byHighByte:= InputData[83], byLowByte:=InputData[82] ));  //82-83,反馈代码
	LoopCounter_In:=BYTE_TO_UINT(InputData[84]);						//84,LooperCounter
	InputData86_In:=InputData[86];											//86
	TagPresent_In:=InputData86_In.0;									//86.0,Tag present，标签存在
	HeadNotConnected_In:=InputData86_In.7;					//86.7,HeadNotConnected，读取头未连接
	ReadLength_In := WORD_TO_UINT( MEM.PackBytesToWord(byHighByte:= InputData[89], byLowByte:=InputData[88] ));  //ReadLength,88-89，读取到的长度
	ErrorCode_In := MEM.PackBytesToWord(byHighByte:= InputData[91], byLowByte:=InputData[90] );  //Error Code 90-91，出错代码	
ELSIF ixChannel=2 THEN 
	ResponseCode_In := WORD_TO_UINT( MEM.PackBytesToWord(byHighByte:= InputData[163], byLowByte:=InputData[162] ));  //162-163,反馈代码
	LoopCounter_In:=BYTE_TO_UINT(InputData[164]);						//164,LooperCounter
	InputData166_In:=InputData[166];											//166
	TagPresent_In:=InputData166_In.0;									//166.0,Tag present，标签存在
	HeadNotConnected_In:=InputData166_In.7;					//166.7,HeadNotConnected，读取头未连接
	ReadLength_In := WORD_TO_UINT( MEM.PackBytesToWord(byHighByte:= InputData[169], byLowByte:=InputData[168] ));  //ReadLength,168-169，读取到的长度
	ErrorCode_In := MEM.PackBytesToWord(byHighByte:= InputData[171], byLowByte:=InputData[170] );  //Error Code 170-171，出错代码
ELSIF ixChannel=3 THEN 
	ResponseCode_In := WORD_TO_UINT( MEM.PackBytesToWord(byHighByte:= InputData[243], byLowByte:=InputData[242] ));  //242-243,反馈代码
	LoopCounter_In:=BYTE_TO_UINT(InputData[244]);						//244,LooperCounter
	InputData6_In:=InputData[246];											//246
	TagPresent_In:=InputData246_In.0;									//246.0,Tag present，标签存在
	HeadNotConnected_In:=InputData246_In.7;					//246.7,HeadNotConnected，读取头未连接
	ReadLength_In := WORD_TO_UINT( MEM.PackBytesToWord(byHighByte:= InputData[249], byLowByte:=InputData[248] ));  //ReadLength,248-249，读取到的长度
	ErrorCode_In := MEM.PackBytesToWord(byHighByte:= InputData[251], byLowByte:=InputData[250] );  //Error Code 250-251，出错代码
ELSE
	 wError:=2;// error，Invalid Parameter -> check the Channel setting
END_IF;

rR_TRIG[0](CLK:=ixRead);		//Read
rR_TRIG[1](CLK:=ixWrite);	//Write
rR_TRIG[2](CLK:=ixReset);	//Reset
//Excute the Command，触发
IF (rR_TRIG[0].Q AND NOT bOldRead) OR (rR_TRIG[1].Q AND NOT bOldWrite)  OR (rR_TRIG[2].Q AND xError) THEN
	IF ixRead THEN OperationType:=16#2;
	ELSIF ixWrite THEN OperationType:=16#4;
	ELSIF ixReset THEN OperationType:=16#8000;
	END_IF;
    bExcute:=TRUE;
END_IF;
//Reset b,复位
IF xError AND ixReset THEN
	wError:=0;
	xBusy:=FALSE;
	iCommandSeq:=0;
END_IF;

//自动流程
CASE iCommandSeq OF
	0:  //Idle Command and Reset Done ，等待触发
	  xDone:=FALSE; //Reset Done marker
      CommandCode_Out:=0;  //Clear the Command
	  IF ResponseCode_In=0 AND LoopCounter_Out=16#0  
		  AND bExcute THEN 
       iCommandSeq:=10;   
	  END_IF;
	  
	 5:	//Clear the Read data，读取前清零接收数据
	  IF ixRead THEN
		  FOR iCnt01:=0 TO 127 BY 1 DO  
				xarbRxData[iCnt01]:=0;	//读取前清零
		  END_FOR;
	  END_IF;
	  iCommandSeq:=10;
	    
	10:  //waiting for Excute start, Then Initial the Command ，执行触发
	     xuiDataLength:=0; //Clear the read data length of FB output
		  //Read Command
			IF ErrorCode_In=0 AND OperationType=16#2 AND OperationType<>16#4 THEN 	
				DataLength_Out:=uiDataLength;//	写入长度
				CommandCode_Out:=16#2;  //read command，读取代码2	
				bExcute:=FALSE;
				iCommandSeq:=20;
			END_IF;
			//Write Command
			IF ErrorCode_In=0 AND OperationType<>16#2 AND OperationType=16#4 THEN 			
				IF ixChannel=0 THEN 		//写入数据更新
					FOR Index2:=0 TO 55 BY 1 DO
						OutputData[Index2+26]:=iarbDataTx[0+Index2];
					END_FOR;	
				ELSIF ixChannel=1 THEN 
					FOR Index2:=0 TO 55 BY 1 DO
						OutputData[Index2+106]:=iarbDataTx[0+Index2];
					END_FOR;
				ELSIF ixChannel=2 THEN 
					FOR Index2:=0 TO 55 BY 1 DO
						OutputData[Index2+186]:=iarbDataTx[0+Index2];
					END_FOR;					
				ELSIF ixChannel=3 THEN 
					FOR Index2:=0 TO 55 BY 1 DO
						OutputData[Index2+266]:=iarbDataTx[0+Index2];
					END_FOR;					
				END_IF;		
				DataLength_Out:=uiDataLength;//	写入长度
				CommandCode_Out:=16#4;  //write command，写入代码4
				bExcute:=FALSE;
				iCommandSeq:=20;
			END_IF;
			//Reset Command
			IF  OperationType=16#8000 AND ErrorCode_In<>0 THEN
				CommandCode_Out:=16#8000 ;  //Reset command，复位代码，16#8000
				bExcute:=FALSE;
				iCommandSeq:=20;
			END_IF	;

	20: //Excuting the Command ,Wait the response from RFID，等待RFID执行
	  IF ResponseCode_In<=0 THEN 
	     xBusy:=TRUE;
	  END_IF;
	   //Command excuting done,No error
      IF ResponseCode_In>0 AND ErrorCode_In=0  THEN 
		  xBusy:=FALSE;
		 iCommandSeq:=30; 
	  END_IF;
	  //Command excuting Done, error occurs
	  IF  ErrorCode_In<>0 THEN 
		 xBusy:=FALSE; 
	  END_IF;
	  
	30: //Set Command Done signal when no error and Deal with Read data，执行完成，触发信号复位后回到0步
		IF  ResponseCode_In<16#4000 
		THEN
		   xDone:=TRUE;
		   xuiDataLength:=ReadLength_In;  //Display of the length of the read data
		   //Read Command Done, Store data from Input mappping
		   IF ResponseCode_In=16#2 THEN 	//读取数据转存
				IF ixChannel=0 THEN 
					FOR Index1:=0 TO 55 BY 1 DO
						xarbRxData[Index1]:=InputData[Index1+26];
					END_FOR;	
				ELSIF ixChannel=1 THEN 
					FOR Index1:=0 TO 55 BY 1 DO
						xarbRxData[Index1]:=InputData[Index1+106];
					END_FOR;
				ELSIF ixChannel=2 THEN 
					FOR Index1:=0 TO 55 BY 1 DO
						xarbRxData[Index1]:=InputData[Index1+186];
					END_FOR;					
				ELSIF ixChannel=3 THEN 
					FOR Index1:=0 TO 55 BY 1 DO
						xarbRxData[Index1]:=InputData[Index1+266];
					END_FOR;					
					
				END_IF;
		   END_IF ;
		 END_IF;
		 IF NOT ixRead AND NOT ixWrite THEN	//触发信号复位后回到0步
	    	iCommandSeq:=0; 
		 END_IF;
END_CASE;

(*Error information*)
IF ixRead AND ixWrite THEN 
	wError:=3;// error，Read and Write are both on，读写同时执行报错
END_IF;

tTimout(IN:=xBusy,PT:=T#3S);  
IF tTimout.Q THEN 
   wError:=1;	           //Timeout for command excuting，超时
END_IF;

(*Function Block output*)
//Error code
IF wError<>0 THEN 
	eErrorCode:=wError;  //Self defined error,自定义报错代码
 ELSE
	eErrorCode:= ErrorCode_In; //Error from RFID，RFID报错代码
 END_IF;
 
//total Error
IF eErrorCode>0 THEN //输出报错
	xError:=TRUE;
 ELSE
	xError:=FALSE;	
END_IF;

xTP:=TagPresent_In;  //Tag Present Status，标签存在输出
xRWHeadNotConnected:=HeadNotConnected_In; //RWHead Connected Status，读头未连接输出
(*Tag UID  information*)
 IF TagPresent_In AND NOT bOldTagPresent AND CommandCode_Out=0 THEN 	//uid输出
	FOR iCnt02:=0 TO 7 BY 1 DO 
	   xarbTagUID[iCnt02]:= InputData[iCnt02];
	END_FOR;
END_IF;
IF bOldTagPresent AND NOT TagPresent_In THEN        //Clear Tag UID information，清除UID
	FOR iCnt02:=0 TO 7 BY 1 DO 
	   xarbTagUID[iCnt02]:= 0 ;
   END_FOR;
END_IF;
(*Controll mapping *)
//WriteLength_Out:=uiDataLength; //Write data length
StartAddress_Out:=UDINT_TO_DWORD( udiStartAddress);   //起始地址
LoopCounter_Out:=0;   //no less than 112 byte per the tag

(*Output mapping*)
IF ixChannel=0 THEN 
	OutputData[4]:=UINT_TO_BYTE( LoopCounter_Out);														//LoopCounter,4
	fbUnpackDWord(
	dwValue:= StartAddress_Out,  
	byLLByte=> OutputData[6], 
	byLHByte=> OutputData[7], 
	byHLByte=> OutputData[8],  
	byHHByte=> OutputData[9], );                                                        //StartAddress,6-9，起始地址
	fbUnpackWord(
	wValue:= UINT_TO_WORD(DataLength_Out), 
	byLowByte=> OutputData[10], 
	byHighByte=> OutputData[11], );                                                     //WriteLength,10-11，写入长度
	fbUnpackWord(
	wValue:= INT_TO_WORD(CommandCode_Out), 
	byLowByte=> OutputData[2], 
	byHighByte=> OutputData[3], );                                                     ///CommandCode,2-3，命令代码
ELSIF ixChannel=1 THEN 
	OutputData[84]:=UINT_TO_BYTE(LoopCounter_Out);														//LoopCounter,84
	fbUnpackDWord(
	dwValue:= StartAddress_Out,  
	byLLByte=> OutputData[86], 
	byLHByte=> OutputData[87], 
	byHLByte=> OutputData[88],  
	byHHByte=> OutputData[89], );                                                        //StartAddress,86-89，起始地址
	fbUnpackWord(
	wValue:= UINT_TO_WORD(DataLength_Out), 
	byLowByte=> OutputData[90], 
	byHighByte=> OutputData[91], );                                                     //WriteLength,90-91，写入长度
	fbUnpackWord(
	wValue:= INT_TO_WORD(CommandCode_Out), 
	byLowByte=> OutputData[82], 
	byHighByte=> OutputData[83], );                                                     ///CommandCode,82-83，命令代码
ELSIF ixChannel=2 THEN 
	OutputData[164]:=UINT_TO_BYTE( LoopCounter_Out);	//LoopCounter,164
		fbUnpackDWord(
	dwValue:= StartAddress_Out,  
	byLLByte=> OutputData[166], 
	byLHByte=> OutputData[167], 
	byHLByte=> OutputData[168],  
	byHHByte=> OutputData[169], );                                                        //StartAddress,166-169，起始地址
	fbUnpackWord(
	wValue:= UINT_TO_WORD(DataLength_Out), 
	byLowByte=> OutputData[170], 
	byHighByte=> OutputData[171], );                                                     //WriteLength,170-171，写入长度
	fbUnpackWord(
	wValue:= INT_TO_WORD(CommandCode_Out), 
	byLowByte=> OutputData[162], 
	byHighByte=> OutputData[163], );                                                     ///CommandCode,162-163，命令代码
ELSIF ixChannel=3 THEN 
	OutputData[244]:=UINT_TO_BYTE( LoopCounter_Out);	//LoopCounter,244
		fbUnpackDWord(
	dwValue:= StartAddress_Out,  
	byLLByte=> OutputData[246], 
	byLHByte=> OutputData[247], 
	byHLByte=> OutputData[248],  
	byHHByte=> OutputData[249], );                                                        //StartAddress,246-249，起始地址
	fbUnpackWord(
	wValue:= UINT_TO_WORD(DataLength_Out), 
	byLowByte=> OutputData[250], 
	byHighByte=> OutputData[251], );                                                     //WriteLength,250-251，写入长度
	fbUnpackWord(
	wValue:= INT_TO_WORD(CommandCode_Out), 
	byLowByte=> OutputData[242], 
	byHighByte=> OutputData[243], );                                                     ///CommandCode,242-243，命令代码
ELSE
	 wError:=2;// error，Invalid Parameter -> check the Channel setting
END_IF;

(* Read and Write old Status*)
bOldRead:=ixRead;
bOldWrite:=ixWrite;
bOldTagPresent:=TagPresent_In;

END_FUNCTION_BLOCK

// ---- Standard/Public/03 HMI/FB_TurnPages_RD.TcPOU
FUNCTION_BLOCK FB_TurnPages_RD
VAR_IN_OUT
IN          : UDT_TurnPages_RD;
END_VAR
VAR_OUTPUT
value       : INT;
change      : BOOL;
END_VAR
VAR
click       : FB_Click_RD;
emptyWord   : WORD;
pos         : UINT;
arypageNumberDisplay : ARRAY[0..15] OF BOOL;
END_VAR

  //================================================================================== 
  // Harmontromics / (C) Copyright (2022) 
  //----------------------------------------------------------------------------------
  // Title:               翻页控制
  // Comment/Function:    上/下一页按钮改变值
  //                      值的范围 minValue <= value <= (maxValue-1)/increment*increment
  //                      value > minValue 时上一页按钮显示
  //                      value < maxValue - increment 时下一页按钮显示                  
  // Library/Family:      (that the source is dedicated to)
  // Author:              David.Wong
  // Target System: 
  // Engineering:          Sysmac Studio
  // Restrictions:        	(OB types, etc.)
  // Requirements:        (hardware, technological package, etc.) 
  //----------------------------------------------------------------------------------
  // Change log table:
  // Version     | Date       | Expert in charge | Changes applied
  //-------------|------------|------------------|------------------------------------
  // 001.000.000 | 2023-8-2  | David.Wong       | First released version
  //             |            |                  |  
  //             |            |                  |              
  //             |            |                  | 
  //================================================================================== 
  
click(CLK := IN.prevClick OR IN.nextClick);
IF click.Q OR value <> IN.value THEN
	IF IN.prevClick AND IN.prevDisplay THEN
		IN.value := IN.value - IN.increment;
	ELSIF IN.nextClick AND IN.nextDisplay THEN
		IN.value := IN.value + IN.increment;
	END_IF;
END_IF;
IN.value := LIMIT(IN.value,IN.minValue,DINT_TO_INT(IN.maxValue / IN.increment * IN.increment));
IN.prevDisplay := IN.value > IN.minValue;
IN.nextDisplay := IN.value < IN.maxValue - IN.increment;
change	:=value <> IN.value;
value := IN.value;
IN.pageNumberDisplay:=emptyWord;
arypageNumberDisplay:=FUN_WordToAry(in:=IN.pageNumberDisplay);
arypageNumberDisplay[INT_TO_USINT((IN.maxValue -IN.minValue) / IN.increment)]:=TRUE;
IN.pageNumberDisplay:=FUN_AryToWord_RD(IN:=arypageNumberDisplay);

END_FUNCTION_BLOCK

// ---- Standard/Unit/00 General/FB_Click_RD.TcPOU
FUNCTION_BLOCK FB_Click_RD
VAR_INPUT
CLK          : BOOL;
END_VAR
VAR_OUTPUT
Q            : BOOL;
END_VAR
VAR
timeCache    : UDINT;
cache        : BOOL;
clickTimer   : TON;
END_VAR

